LIN {X 0,Y 305.442,Z 224.06,A -85,B 0,C 180,E1 -15871.952,E2 -15871.952} C_VEL
LIN {X 0,Y 305.457,Z 224.06,A -85,B 0,C 180,E1 -15875.114,E2 -15875.114} C_VEL
LIN {X 0,Y 305.461,Z 224.056,A -85,B 0,C 180,E1 -15878.533,E2 -15878.533} C_VEL
LIN {X 0,Y 305.45,Z 224.057,A -85,B 0,C 180,E1 -15882.586,E2 -15882.586} C_VEL
LIN {X 0,Y 305.451,Z 224.223,A -85,B 0,C 180,E1 -15887.041,E2 -15887.041} C_VEL
LIN {X 0,Y 308.59,Z 234.406,A -85,B 0,C 180,E1 -15890.382,E2 -15890.382} C_VEL
LIN {X 0,Y 309.647,Z 238.195,A -85,B 0,C 180,E1 -15891.521,E2 -15891.521} C_VEL
LIN {X 0,Y 318.972,Z 255.957,A -85,B 0,C 180,E1 -15893.321,E2 -15893.321} C_VEL
LIN {X 0,Y 327.178,Z 273.763,A -85,B 0,C 180,E1 -15894.846,E2 -15894.846} C_VEL
LIN {X 0,Y 329.476,Z 279.574,A -85,B 0,C 180,E1 -15895.276,E2 -15895.276} C_VEL
LIN {X 0,Y 331.457,Z 291.54,A -85,B 0,C 180,E1 -15895.818,E2 -15895.818} C_VEL
LIN {X 0,Y 327.97,Z 393.454,A -85,B 0,C 180,E1 -15898.016,E2 -15898.016} C_VEL
LIN {X 0,Y 327.096,Z 410.423,A -85,B 0,C 180,E1 -15898.464,E2 -15898.464} C_VEL
LIN {X 0,Y 325.725,Z 425.453,A -85,B 0,C 180,E1 -15899.084,E2 -15899.084} C_VEL
LIN {X 0,Y 323.988,Z 439.556,A -85,B 0,C 180,E1 -15899.893,E2 -15899.893} C_VEL
LIN {X 0,Y 321.936,Z 453.745,A -85,B 0,C 180,E1 -15900.966,E2 -15900.966} C_VEL
LIN {X 0,Y 319.46,Z 467.76,A -85,B 0,C 180,E1 -15902.307,E2 -15902.307} C_VEL
LIN {X 0,Y 316.903,Z 480.688,A -85,B 0,C 180,E1 -15903.848,E2 -15903.848} C_VEL
LIN {X 0,Y 314.412,Z 492.531,A -85,B 0,C 180,E1 -15905.574,E2 -15905.574} C_VEL
LIN {X 0,Y 311.997,Z 503.387,A -85,B 0,C 180,E1 -15907.485,E2 -15907.485} C_VEL
LIN {X 0,Y 309.684,Z 513.966,A -85,B 0,C 180,E1 -15909.752,E2 -15909.752} C_VEL
LIN {X 0,Y 307.669,Z 522.772,A -85,B 0,C 180,E1 -15912.039,E2 -15912.039} C_VEL
LIN {X 0,Y 306.367,Z 529.155,A -85,B 0,C 180,E1 -15914.022,E2 -15914.022} C_VEL
LIN {X 0,Y 305.081,Z 536.165,A -85,B 0,C 180,E1 -15916.682,E2 -15916.682} C_VEL
LIN {X 0,Y 304.17,Z 541.679,A -85,B 0,C 180,E1 -15919.348,E2 -15919.348} C_VEL
LIN {X 0,Y 303.765,Z 545.855,A -85,B 0,C 180,E1 -15922.021,E2 -15922.021} C_VEL
LIN {X 0,Y 303.596,Z 548.785,A -85,B 0,C 180,E1 -15924.687,E2 -15924.687} C_VEL
LIN {X 0,Y 303.59,Z 550.533,A -85,B 0,C 180,E1 -15927.346,E2 -15927.346} C_VEL
LIN {X 0,Y 303.602,Z 551.13,A -85,B 0,C 180,E1 -15930,E2 -15930} C_VEL
LIN {X 0,Y 303.59,Z 550.523,A -85,B 0,C 180,E1 -15932.654,E2 -15932.654} C_VEL
LIN {X 0,Y 303.624,Z 548.564,A -85,B 0,C 180,E1 -15935.544,E2 -15935.544} C_VEL
LIN {X 0,Y 303.765,Z 545.825,A -85,B 0,C 180,E1 -15937.979,E2 -15937.979} C_VEL
LIN {X 0,Y 304.169,Z 541.644,A -85,B 0,C 180,E1 -15940.652,E2 -15940.652} C_VEL
LIN {X 0,Y 305.068,Z 536.114,A -85,B 0,C 180,E1 -15943.319,E2 -15943.319} C_VEL
LIN {X 0,Y 306.353,Z 529.083,A -85,B 0,C 180,E1 -15945.979,E2 -15945.979} C_VEL
LIN {X 0,Y 308.205,Z 520.343,A -85,B 0,C 180,E1 -15948.617,E2 -15948.617} C_VEL
LIN {X 0,Y 310.329,Z 511.066,A -85,B 0,C 180,E1 -15950.897,E2 -15950.897} C_VEL
LIN {X 0,Y 312.328,Z 501.805,A -85,B 0,C 180,E1 -15952.804,E2 -15952.804} C_VEL
LIN {X 0,Y 314.818,Z 490.441,A -85,B 0,C 180,E1 -15954.744,E2 -15954.744} C_VEL
LIN {X 0,Y 317.361,Z 478.179,A -85,B 0,C 180,E1 -15956.466,E2 -15956.466} C_VEL
LIN {X 0,Y 320.016,Z 464.701,A -85,B 0,C 180,E1 -15957.996,E2 -15957.996} C_VEL
LIN {X 0,Y 322.473,Z 449.936,A -85,B 0,C 180,E1 -15959.336,E2 -15959.336} C_VEL
LIN {X 0,Y 324.543,Z 434.588,A -85,B 0,C 180,E1 -15960.409,E2 -15960.409} C_VEL
LIN {X 0,Y 326.232,Z 419.535,A -85,B 0,C 180,E1 -15961.178,E2 -15961.178} C_VEL
LIN {X 0,Y 327.477,Z 403.763,A -85,B 0,C 180,E1 -15961.721,E2 -15961.721} C_VEL
LIN {X 0,Y 331.104,Z 302.228,A -85,B 0,C 180,E1 -15963.922,E2 -15963.922} C_VEL
LIN {X 0,Y 331.324,Z 291.096,A -85,B 0,C 180,E1 -15964.182,E2 -15964.182} C_VEL
LIN {X 0,Y 328.976,Z 277.875,A -85,B 0,C 180,E1 -15964.8,E2 -15964.8} C_VEL
LIN {X 0,Y 319.974,Z 258.117,A -85,B 0,C 180,E1 -15966.456,E2 -15966.456} C_VEL
LIN {X 0,Y 313.704,Z 245.865,A -85,B 0,C 180,E1 -15967.645,E2 -15967.645} C_VEL
LIN {X 0,Y 309.583,Z 237.999,A -85,B 0,C 180,E1 -15968.468,E2 -15968.468} C_VEL
LIN {X 0,Y 306.264,Z 226.625,A -85,B 0,C 180,E1 -15972.098,E2 -15972.098} C_VEL
LIN {X 0,Y 305.447,Z 224.059,A -85,B 0,C 180,E1 -15972.977,E2 -15972.977} C_VEL
LIN {X 0,Y 305.474,Z 224.053,A -85,B 0,C 180,E1 -15977.409,E2 -15977.409} C_VEL
LIN {X 0,Y 305.504,Z 224.047,A -85,B 0,C 180,E1 -15981.602,E2 -15981.602} C_VEL
LIN {X 0,Y 305.458,Z 224.052,A -85,B 0,C 180,E1 -15984.886,E2 -15984.886} C_VEL
LIN {X 0,Y 305.451,Z 224.059,A -85,B 0,C 180,E1 -15988.353,E2 -15988.353} C_VEL
LIN {X 0,Y 305.523,Z 224.048,A -85,B 0,C 180,E1 -15991.114,E2 -15991.114} C_VEL
LIN {X 0,Y 305.565,Z 224.045,A -85,B 0,C 180,E1 -15994.088,E2 -15994.088} C_VEL
LIN {X 0,Y 305.466,Z 224.029,A -85,B 0,C 180,E1 -15998.4,E2 -15998.4} C_VEL
LIN {X 0,Y 305.583,Z 224.043,A -85,B 0,C 180,E1 -16001.217,E2 -16001.217} C_VEL
LIN {X 0,Y 305.642,Z 224.038,A -85,B 0,C 180,E1 -16005.349,E2 -16005.349} C_VEL
LIN {X 0,Y 305.629,Z 224.041,A -85,B 0,C 180,E1 -16009.4,E2 -16009.4} C_VEL
LIN {X 0,Y 305.79,Z 224.013,A -85,B 0,C 180,E1 -16012.074,E2 -16012.074} C_VEL
LIN {X 0,Y 305.68,Z 224.031,A -85,B 0,C 180,E1 -16014.723,E2 -16014.723} C_VEL
LIN {X 0,Y 305.952,Z 223.998,A -85,B 0,C 180,E1 -16018.684,E2 -16018.684} C_VEL
LIN {X 0,Y 305.952,Z 223.996,A -85,B 0,C 180,E1 -16021.316,E2 -16021.316} C_VEL
LIN {X 0,Y 305.836,Z 224.013,A -85,B 0,C 180,E1 -16026.6,E2 -16026.6} C_VEL
LIN {X 0,Y 305.698,Z 224.024,A -85,B 0,C 180,E1 -16029.261,E2 -16029.261} C_VEL
LIN {X 0,Y 305.582,Z 224.039,A -85,B 0,C 180,E1 -16033.296,E2 -16033.296} C_VEL
LIN {X 0,Y 305.587,Z 224.04,A -85,B 0,C 180,E1 -16036.021,E2 -16036.021} C_VEL
LIN {X 0,Y 305.554,Z 224.047,A -85,B 0,C 180,E1 -16039.436,E2 -16039.436} C_VEL
LIN {X 0,Y 305.481,Z 224.058,A -85,B 0,C 180,E1 -16043.04,E2 -16043.04} C_VEL
LIN {X 0,Y 305.521,Z 224.021,A -85,B 0,C 180,E1 -16046.219,E2 -16046.219} C_VEL
LIN {X 0,Y 305.491,Z 224.057,A -85,B 0,C 180,E1 -16049.051,E2 -16049.051} C_VEL
LIN {X 0,Y 305.46,Z 224.055,A -85,B 0,C 180,E1 -16053.518,E2 -16053.518} C_VEL
LIN {X 0,Y 305.471,Z 224.053,A -85,B 0,C 180,E1 -16056.74,E2 -16056.74} C_VEL
LIN {X 0,Y 305.451,Z 224.059,A -85,B 0,C 180,E1 -16060.6,E2 -16060.6} C_VEL
LIN {X 0,Y 305.416,Z 224.061,A -85,B 0,C 180,E1 -16064.493,E2 -16064.493} C_VEL
LIN {X 0,Y 305.44,Z 224.062,A -85,B 0,C 180,E1 -16068.144,E2 -16068.144} C_VEL
LIN {X 0,Y 305.483,Z 224.145,A -85,B 0,C 180,E1 -16070.766,E2 -16070.766} C_VEL
LIN {X 0,Y 305.611,Z 224.87,A -85,B 0,C 180,E1 -16071.007,E2 -16071.007} C_VEL
LIN {X 0,Y 306.861,Z 227.498,A -85,B 0,C 180,E1 -16071.275,E2 -16071.275} C_VEL
LIN {X 0,Y 309.527,Z 231.534,A -85,B 0,C 180,E1 -16071.79,E2 -16071.79} C_VEL
LIN {X 0,Y 317.49,Z 245.518,A -85,B 0,C 180,E1 -16073.31,E2 -16073.31} C_VEL
LIN {X 0,Y 326.019,Z 262.428,A -85,B 0,C 180,E1 -16074.876,E2 -16074.876} C_VEL
LIN {X 0,Y 331.826,Z 275.27,A -85,B 0,C 180,E1 -16075.915,E2 -16075.915} C_VEL
LIN {X 0,Y 329.059,Z 358.793,A -85,B 0,C 180,E1 -16077.728,E2 -16077.728} C_VEL
LIN {X 0,Y 327.79,Z 390.563,A -85,B 0,C 180,E1 -16078.448,E2 -16078.448} C_VEL
LIN {X 0,Y 326.666,Z 405.546,A -85,B 0,C 180,E1 -16079.012,E2 -16079.012} C_VEL
LIN {X 0,Y 325.15,Z 420.181,A -85,B 0,C 180,E1 -16079.804,E2 -16079.804} C_VEL
LIN {X 0,Y 323.55,Z 433.262,A -85,B 0,C 180,E1 -16080.75,E2 -16080.75} C_VEL
LIN {X 0,Y 321.4,Z 446.754,A -85,B 0,C 180,E1 -16081.958,E2 -16081.958} C_VEL
LIN {X 0,Y 318.907,Z 460.516,A -85,B 0,C 180,E1 -16083.496,E2 -16083.496} C_VEL
LIN {X 0,Y 316.328,Z 473.036,A -85,B 0,C 180,E1 -16085.224,E2 -16085.224} C_VEL
LIN {X 0,Y 314.517,Z 481.644,A -85,B 0,C 180,E1 -16086.652,E2 -16086.652} C_VEL
LIN {X 0,Y 312.254,Z 491.48,A -85,B 0,C 180,E1 -16088.547,E2 -16088.547} C_VEL
LIN {X 0,Y 310.028,Z 501.175,A -85,B 0,C 180,E1 -16090.811,E2 -16090.811} C_VEL
LIN {X 0,Y 308.029,Z 509.515,A -85,B 0,C 180,E1 -16093.177,E2 -16093.177} C_VEL
LIN {X 0,Y 306.709,Z 515.914,A -85,B 0,C 180,E1 -16095.401,E2 -16095.401} C_VEL
LIN {X 0,Y 305.37,Z 522.081,A -85,B 0,C 180,E1 -16098.046,E2 -16098.046} C_VEL
LIN {X 0,Y 304.567,Z 526.836,A -85,B 0,C 180,E1 -16100.705,E2 -16100.705} C_VEL
LIN {X 0,Y 304.046,Z 530.318,A -85,B 0,C 180,E1 -16103.363,E2 -16103.363} C_VEL
LIN {X 0,Y 303.786,Z 532.618,A -85,B 0,C 180,E1 -16106.02,E2 -16106.02} C_VEL
LIN {X 0,Y 303.608,Z 533.793,A -85,B 0,C 180,E1 -16108.674,E2 -16108.674} C_VEL
LIN {X 0,Y 303.608,Z 533.807,A -85,B 0,C 180,E1 -16111.326,E2 -16111.326} C_VEL
LIN {X 0,Y 303.781,Z 532.688,A -85,B 0,C 180,E1 -16113.98,E2 -16113.98} C_VEL
LIN {X 0,Y 304.041,Z 530.442,A -85,B 0,C 180,E1 -16116.637,E2 -16116.637} C_VEL
LIN {X 0,Y 304.551,Z 527.011,A -85,B 0,C 180,E1 -16119.296,E2 -16119.296} C_VEL
LIN {X 0,Y 305.342,Z 522.312,A -85,B 0,C 180,E1 -16121.955,E2 -16121.955} C_VEL
LIN {X 0,Y 306.689,Z 516.215,A -85,B 0,C 180,E1 -16124.6,E2 -16124.6} C_VEL
LIN {X 0,Y 308.303,Z 508.54,A -85,B 0,C 180,E1 -16127.238,E2 -16127.238} C_VEL
LIN {X 0,Y 310.234,Z 500.35,A -85,B 0,C 180,E1 -16129.52,E2 -16129.52} C_VEL
LIN {X 0,Y 312.498,Z 490.48,A -85,B 0,C 180,E1 -16131.782,E2 -16131.782} C_VEL
LIN {X 0,Y 314.726,Z 480.279,A -85,B 0,C 180,E1 -16133.715,E2 -16133.715} C_VEL
LIN {X 0,Y 317.374,Z 468.298,A -85,B 0,C 180,E1 -16135.582,E2 -16135.582} C_VEL
LIN {X 0,Y 319.711,Z 456.205,A -85,B 0,C 180,E1 -16137.137,E2 -16137.137} C_VEL
LIN {X 0,Y 322.091,Z 443.055,A -85,B 0,C 180,E1 -16138.509,E2 -16138.509} C_VEL
LIN {X 0,Y 323.994,Z 429.914,A -85,B 0,C 180,E1 -16139.624,E2 -16139.624} C_VEL
LIN {X 0,Y 325.759,Z 415.327,A -85,B 0,C 180,E1 -16140.589,E2 -16140.589} C_VEL
LIN {X 0,Y 327.093,Z 400.58,A -85,B 0,C 180,E1 -16141.311,E2 -16141.311} C_VEL
LIN {X 0,Y 328.13,Z 385.845,A -85,B 0,C 180,E1 -16141.786,E2 -16141.786} C_VEL
LIN {X 0,Y 331.438,Z 291.969,A -85,B 0,C 180,E1 -16143.82,E2 -16143.82} C_VEL
LIN {X 0,Y 331.228,Z 288.126,A -85,B 0,C 180,E1 -16143.943,E2 -16143.943} C_VEL
LIN {X 0,Y 329.748,Z 282.696,A -85,B 0,C 180,E1 -16144.258,E2 -16144.258} C_VEL
LIN {X 0,Y 327.401,Z 277.728,A -85,B 0,C 180,E1 -16144.67,E2 -16144.67} C_VEL
LIN {X 0,Y 323.608,Z 271.295,A -85,B 0,C 180,E1 -16145.31,E2 -16145.31} C_VEL
LIN {X 0,Y 320.146,Z 264.635,A -85,B 0,C 180,E1 -16145.934,E2 -16145.934} C_VEL
LIN {X 0,Y 311.45,Z 247.476,A -85,B 0,C 180,E1 -16147.599,E2 -16147.599} C_VEL
LIN {X 0,Y 304.686,Z 235.632,A -85,B 0,C 180,E1 -16148.943,E2 -16148.943} C_VEL
LIN {X 0,Y 300.541,Z 229.139,A -85,B 0,C 180,E1 -16149.786,E2 -16149.786} C_VEL
LIN {X 0,Y 298.891,Z 226.755,A -85,B 0,C 180,E1 -16150.126,E2 -16150.126} C_VEL
LIN {X 0,Y 298.433,Z 224.941,A -85,B 0,C 180,E1 -16150.304,E2 -16150.304} C_VEL
LIN {X 0,Y 298.396,Z 224.942,A -85,B 0,C 180,E1 -16153.102,E2 -16153.102} C_VEL
LIN {X 0,Y 298.4,Z 224.925,A -85,B 0,C 180,E1 -16156.92,E2 -16156.92} C_VEL
LIN {X 0,Y 298.421,Z 224.928,A -85,B 0,C 180,E1 -16161,E2 -16161} C_VEL
LIN {X 0,Y 298.428,Z 224.923,A -85,B 0,C 180,E1 -16163.931,E2 -16163.931} C_VEL
LIN {X 0,Y 298.39,Z 224.913,A -85,B 0,C 180,E1 -16167.983,E2 -16167.983} C_VEL
LIN {X 0,Y 298.459,Z 224.933,A -85,B 0,C 180,E1 -16171.904,E2 -16171.904} C_VEL
LIN {X 0,Y 298.48,Z 224.928,A -85,B 0,C 180,E1 -16174.923,E2 -16174.923} C_VEL
LIN {X 0,Y 298.444,Z 224.936,A -85,B 0,C 180,E1 -16179.315,E2 -16179.315} C_VEL
LIN {X 0,Y 298.531,Z 224.916,A -85,B 0,C 180,E1 -16182.179,E2 -16182.179} C_VEL
LIN {X 0,Y 298.587,Z 224.908,A -85,B 0,C 180,E1 -16184.994,E2 -16184.994} C_VEL
LIN {X 0,Y 298.587,Z 224.911,A -85,B 0,C 180,E1 -16189.146,E2 -16189.146} C_VEL
LIN {X 0,Y 298.748,Z 224.895,A -85,B 0,C 180,E1 -16191.886,E2 -16191.886} C_VEL
LIN {X 0,Y 298.651,Z 224.899,A -85,B 0,C 180,E1 -16194.599,E2 -16194.599} C_VEL
LIN {X 0,Y 298.918,Z 224.867,A -85,B 0,C 180,E1 -16198.653,E2 -16198.653} C_VEL
LIN {X 0,Y 298.918,Z 224.875,A -85,B 0,C 180,E1 -16201.347,E2 -16201.347} C_VEL
LIN {X 0,Y 298.78,Z 224.893,A -85,B 0,C 180,E1 -16206.754,E2 -16206.754} C_VEL
LIN {X 0,Y 298.629,Z 224.908,A -85,B 0,C 180,E1 -16209.482,E2 -16209.482} C_VEL
LIN {X 0,Y 298.545,Z 224.916,A -85,B 0,C 180,E1 -16213.616,E2 -16213.616} C_VEL
LIN {X 0,Y 298.542,Z 224.919,A -85,B 0,C 180,E1 -16216.409,E2 -16216.409} C_VEL
LIN {X 0,Y 298.506,Z 224.93,A -85,B 0,C 180,E1 -16219.655,E2 -16219.655} C_VEL
LIN {X 0,Y 298.451,Z 224.936,A -85,B 0,C 180,E1 -16223.598,E2 -16223.598} C_VEL
LIN {X 0,Y 298.484,Z 224.927,A -85,B 0,C 180,E1 -16226.575,E2 -16226.575} C_VEL
LIN {X 0,Y 298.417,Z 224.94,A -85,B 0,C 180,E1 -16229.641,E2 -16229.641} C_VEL
LIN {X 0,Y 298.392,Z 224.932,A -85,B 0,C 180,E1 -16232.8,E2 -16232.8} C_VEL
LIN {X 0,Y 298.446,Z 224.929,A -85,B 0,C 180,E1 -16236.809,E2 -16236.809} C_VEL
LIN {X 0,Y 298.404,Z 224.918,A -85,B 0,C 180,E1 -16239.487,E2 -16239.487} C_VEL
LIN {X 0,Y 298.395,Z 224.942,A -85,B 0,C 180,E1 -16243.104,E2 -16243.104} C_VEL
LIN {X 0,Y 298.394,Z 225.075,A -85,B 0,C 180,E1 -16246.1,E2 -16246.1} C_VEL
LIN {X 0,Y 301.445,Z 234.9,A -85,B 0,C 180,E1 -16249.46,E2 -16249.46} C_VEL
LIN {X 0,Y 302.411,Z 238.056,A -85,B 0,C 180,E1 -16250.426,E2 -16250.426} C_VEL
LIN {X 0,Y 310.708,Z 253.532,A -85,B 0,C 180,E1 -16252.116,E2 -16252.116} C_VEL
LIN {X 0,Y 318.046,Z 268.606,A -85,B 0,C 180,E1 -16253.545,E2 -16253.545} C_VEL
LIN {X 0,Y 323.814,Z 281.919,A -85,B 0,C 180,E1 -16254.645,E2 -16254.645} C_VEL
LIN {X 0,Y 325.566,Z 292.715,A -85,B 0,C 180,E1 -16255.147,E2 -16255.147} C_VEL
LIN {X 0,Y 321.912,Z 395.064,A -85,B 0,C 180,E1 -16257.387,E2 -16257.387} C_VEL
LIN {X 0,Y 320.987,Z 411.376,A -85,B 0,C 180,E1 -16257.838,E2 -16257.838} C_VEL
LIN {X 0,Y 319.482,Z 426.787,A -85,B 0,C 180,E1 -16258.504,E2 -16258.504} C_VEL
LIN {X 0,Y 317.701,Z 440.493,A -85,B 0,C 180,E1 -16259.325,E2 -16259.325} C_VEL
LIN {X 0,Y 315.553,Z 454.674,A -85,B 0,C 180,E1 -16260.438,E2 -16260.438} C_VEL
LIN {X 0,Y 313.181,Z 467.563,A -85,B 0,C 180,E1 -16261.703,E2 -16261.703} C_VEL
LIN {X 0,Y 310.492,Z 480.489,A -85,B 0,C 180,E1 -16263.265,E2 -16263.265} C_VEL
LIN {X 0,Y 307.899,Z 492.331,A -85,B 0,C 180,E1 -16265.022,E2 -16265.022} C_VEL
LIN {X 0,Y 305.281,Z 503.599,A -85,B 0,C 180,E1 -16267.051,E2 -16267.051} C_VEL
LIN {X 0,Y 302.994,Z 513.766,A -85,B 0,C 180,E1 -16269.285,E2 -16269.285} C_VEL
LIN {X 0,Y 300.866,Z 522.572,A -85,B 0,C 180,E1 -16271.619,E2 -16271.619} C_VEL
LIN {X 0,Y 299.142,Z 530.594,A -85,B 0,C 180,E1 -16274.234,E2 -16274.234} C_VEL
LIN {X 0,Y 297.851,Z 537.459,A -85,B 0,C 180,E1 -16277.047,E2 -16277.047} C_VEL
LIN {X 0,Y 296.989,Z 542.647,A -85,B 0,C 180,E1 -16279.777,E2 -16279.777} C_VEL
LIN {X 0,Y 296.691,Z 545.654,A -85,B 0,C 180,E1 -16281.829,E2 -16281.829} C_VEL
LIN {X 0,Y 296.511,Z 548.584,A -85,B 0,C 180,E1 -16284.56,E2 -16284.56} C_VEL
LIN {X 0,Y 296.514,Z 550.332,A -85,B 0,C 180,E1 -16287.283,E2 -16287.283} C_VEL
LIN {X 0,Y 296.517,Z 550.93,A -85,B 0,C 180,E1 -16290,E2 -16290} C_VEL
LIN {X 0,Y 296.514,Z 550.322,A -85,B 0,C 180,E1 -16292.717,E2 -16292.717} C_VEL
LIN {X 0,Y 296.511,Z 548.56,A -85,B 0,C 180,E1 -16295.44,E2 -16295.44} C_VEL
LIN {X 0,Y 296.691,Z 545.622,A -85,B 0,C 180,E1 -16298.171,E2 -16298.171} C_VEL
LIN {X 0,Y 297.131,Z 541.44,A -85,B 0,C 180,E1 -16300.907,E2 -16300.907} C_VEL
LIN {X 0,Y 298.079,Z 535.909,A -85,B 0,C 180,E1 -16303.637,E2 -16303.637} C_VEL
LIN {X 0,Y 299.476,Z 528.879,A -85,B 0,C 180,E1 -16306.356,E2 -16306.356} C_VEL
LIN {X 0,Y 301.409,Z 520.138,A -85,B 0,C 180,E1 -16309.052,E2 -16309.052} C_VEL
LIN {X 0,Y 303.648,Z 510.861,A -85,B 0,C 180,E1 -16311.379,E2 -16311.379} C_VEL
LIN {X 0,Y 305.786,Z 501.431,A -85,B 0,C 180,E1 -16313.357,E2 -16313.357} C_VEL
LIN {X 0,Y 308.572,Z 489.208,A -85,B 0,C 180,E1 -16315.46,E2 -16315.46} C_VEL
LIN {X 0,Y 311.268,Z 476.747,A -85,B 0,C 180,E1 -16317.207,E2 -16317.207} C_VEL
LIN {X 0,Y 313.744,Z 464.495,A -85,B 0,C 180,E1 -16318.607,E2 -16318.607} C_VEL
LIN {X 0,Y 316.096,Z 450.844,A -85,B 0,C 180,E1 -16319.875,E2 -16319.875} C_VEL
LIN {X 0,Y 318.272,Z 435.634,A -85,B 0,C 180,E1 -16320.982,E2 -16320.982} C_VEL
LIN {X 0,Y 320.097,Z 420.216,A -85,B 0,C 180,E1 -16321.798,E2 -16321.798} C_VEL
LIN {X 0,Y 321.386,Z 404.975,A -85,B 0,C 180,E1 -16322.348,E2 -16322.348} C_VEL
LIN {X 0,Y 325.197,Z 303.142,A -85,B 0,C 180,E1 -16324.596,E2 -16324.596} C_VEL
LIN {X 0,Y 325.438,Z 292.247,A -85,B 0,C 180,E1 -16324.852,E2 -16324.852} C_VEL
LIN {X 0,Y 323.35,Z 280.676,A -85,B 0,C 180,E1 -16325.416,E2 -16325.416} C_VEL
LIN {X 0,Y 314.797,Z 261.749,A -85,B 0,C 180,E1 -16327.048,E2 -16327.048} C_VEL
LIN {X 0,Y 308.991,Z 250.246,A -85,B 0,C 180,E1 -16328.19,E2 -16328.19} C_VEL
LIN {X 0,Y 302.262,Z 237.669,A -85,B 0,C 180,E1 -16329.597,E2 -16329.597} C_VEL
LIN {X 0,Y 299.227,Z 227.707,A -85,B 0,C 180,E1 -16332.931,E2 -16332.931} C_VEL
LIN {X 0,Y 298.367,Z 224.945,A -85,B 0,C 180,E1 -16333.955,E2 -16333.955} C_VEL
LIN {X 0,Y 298.399,Z 224.934,A -85,B 0,C 180,E1 -16336.92,E2 -16336.92} C_VEL
LIN {X 0,Y 298.421,Z 224.932,A -85,B 0,C 180,E1 -16341.001,E2 -16341.001} C_VEL
LIN {X 0,Y 298.427,Z 224.927,A -85,B 0,C 180,E1 -16343.932,E2 -16343.932} C_VEL
LIN {X 0,Y 298.394,Z 224.934,A -85,B 0,C 180,E1 -16347.982,E2 -16347.982} C_VEL
LIN {X 0,Y 298.463,Z 224.931,A -85,B 0,C 180,E1 -16351.904,E2 -16351.904} C_VEL
LIN {X 0,Y 298.478,Z 224.93,A -85,B 0,C 180,E1 -16354.924,E2 -16354.924} C_VEL
LIN {X 0,Y 298.431,Z 224.911,A -85,B 0,C 180,E1 -16359.314,E2 -16359.314} C_VEL
LIN {X 0,Y 298.531,Z 224.923,A -85,B 0,C 180,E1 -16362.179,E2 -16362.179} C_VEL
LIN {X 0,Y 298.587,Z 224.914,A -85,B 0,C 180,E1 -16364.995,E2 -16364.995} C_VEL
LIN {X 0,Y 298.585,Z 224.916,A -85,B 0,C 180,E1 -16369.146,E2 -16369.146} C_VEL
LIN {X 0,Y 298.734,Z 224.891,A -85,B 0,C 180,E1 -16371.885,E2 -16371.885} C_VEL
LIN {X 0,Y 298.651,Z 224.907,A -85,B 0,C 180,E1 -16374.599,E2 -16374.599} C_VEL
LIN {X 0,Y 298.918,Z 224.875,A -85,B 0,C 180,E1 -16378.653,E2 -16378.653} C_VEL
LIN {X 0,Y 298.918,Z 224.872,A -85,B 0,C 180,E1 -16381.347,E2 -16381.347} C_VEL
LIN {X 0,Y 298.781,Z 224.893,A -85,B 0,C 180,E1 -16386.754,E2 -16386.754} C_VEL
LIN {X 0,Y 298.629,Z 224.906,A -85,B 0,C 180,E1 -16389.482,E2 -16389.482} C_VEL
LIN {X 0,Y 298.545,Z 224.917,A -85,B 0,C 180,E1 -16393.616,E2 -16393.616} C_VEL
LIN {X 0,Y 298.542,Z 224.916,A -85,B 0,C 180,E1 -16396.409,E2 -16396.409} C_VEL
LIN {X 0,Y 298.492,Z 224.925,A -85,B 0,C 180,E1 -16399.647,E2 -16399.647} C_VEL
LIN {X 0,Y 298.423,Z 224.932,A -85,B 0,C 180,E1 -16403.601,E2 -16403.601} C_VEL
LIN {X 0,Y 298.481,Z 224.899,A -85,B 0,C 180,E1 -16406.575,E2 -16406.575} C_VEL
LIN {X 0,Y 298.416,Z 224.937,A -85,B 0,C 180,E1 -16409.642,E2 -16409.642} C_VEL
LIN {X 0,Y 298.391,Z 224.941,A -85,B 0,C 180,E1 -16412.801,E2 -16412.801} C_VEL
LIN {X 0,Y 298.442,Z 224.928,A -85,B 0,C 180,E1 -16416.808,E2 -16416.808} C_VEL
LIN {X 0,Y 298.384,Z 224.938,A -85,B 0,C 180,E1 -16421.089,E2 -16421.089} C_VEL
LIN {X 0,Y 298.386,Z 224.94,A -85,B 0,C 180,E1 -16425.042,E2 -16425.042} C_VEL
LIN {X 0,Y 298.385,Z 224.943,A -85,B 0,C 180,E1 -16428.913,E2 -16428.913} C_VEL
LIN {X 0,Y 298.435,Z 225.115,A -85,B 0,C 180,E1 -16429.881,E2 -16429.881} C_VEL
LIN {X 0,Y 299.537,Z 227.962,A -85,B 0,C 180,E1 -16430.147,E2 -16430.147} C_VEL
LIN {X 0,Y 301.218,Z 230.109,A -85,B 0,C 180,E1 -16430.481,E2 -16430.481} C_VEL
LIN {X 0,Y 308.701,Z 242.483,A -85,B 0,C 180,E1 -16431.986,E2 -16431.986} C_VEL
LIN {X 0,Y 317.512,Z 259.222,A -85,B 0,C 180,E1 -16433.692,E2 -16433.692} C_VEL
LIN {X 0,Y 325.916,Z 277.372,A -85,B 0,C 180,E1 -16435.258,E2 -16435.258} C_VEL
LIN {X 0,Y 323.813,Z 336.928,A -85,B 0,C 180,E1 -16436.566,E2 -16436.566} C_VEL
LIN {X 0,Y 321.857,Z 389.625,A -85,B 0,C 180,E1 -16437.751,E2 -16437.751} C_VEL
LIN {X 0,Y 320.696,Z 404.902,A -85,B 0,C 180,E1 -16438.319,E2 -16438.319} C_VEL
LIN {X 0,Y 319.093,Z 420.18,A -85,B 0,C 180,E1 -16439.153,E2 -16439.153} C_VEL
LIN {X 0,Y 317.329,Z 433.812,A -85,B 0,C 180,E1 -16440.15,E2 -16440.15} C_VEL
LIN {X 0,Y 314.882,Z 448.515,A -85,B 0,C 180,E1 -16441.506,E2 -16441.506} C_VEL
LIN {X 0,Y 312.3,Z 461.969,A -85,B 0,C 180,E1 -16443.071,E2 -16443.071} C_VEL
LIN {X 0,Y 309.636,Z 474.371,A -85,B 0,C 180,E1 -16444.849,E2 -16444.849} C_VEL
LIN {X 0,Y 307.805,Z 482.665,A -85,B 0,C 180,E1 -16446.276,E2 -16446.276} C_VEL
LIN {X 0,Y 305.245,Z 493.161,A -85,B 0,C 180,E1 -16448.384,E2 -16448.384} C_VEL
LIN {X 0,Y 303.007,Z 502.6,A -85,B 0,C 180,E1 -16450.7,E2 -16450.7} C_VEL
LIN {X 0,Y 300.771,Z 511.387,A -85,B 0,C 180,E1 -16453.342,E2 -16453.342} C_VEL
LIN {X 0,Y 299.452,Z 517.786,A -85,B 0,C 180,E1 -16455.734,E2 -16455.734} C_VEL
LIN {X 0,Y 298.134,Z 523.6,A -85,B 0,C 180,E1 -16458.442,E2 -16458.442} C_VEL
LIN {X 0,Y 297.53,Z 527.038,A -85,B 0,C 180,E1 -16460.483,E2 -16460.483} C_VEL
LIN {X 0,Y 296.999,Z 530.519,A -85,B 0,C 180,E1 -16463.205,E2 -16463.205} C_VEL
LIN {X 0,Y 296.703,Z 532.819,A -85,B 0,C 180,E1 -16465.925,E2 -16465.925} C_VEL
LIN {X 0,Y 296.527,Z 533.994,A -85,B 0,C 180,E1 -16468.642,E2 -16468.642} C_VEL
LIN {X 0,Y 296.527,Z 534.008,A -85,B 0,C 180,E1 -16471.358,E2 -16471.358} C_VEL
LIN {X 0,Y 296.697,Z 532.889,A -85,B 0,C 180,E1 -16474.075,E2 -16474.075} C_VEL
LIN {X 0,Y 296.963,Z 530.643,A -85,B 0,C 180,E1 -16476.796,E2 -16476.796} C_VEL
LIN {X 0,Y 297.516,Z 527.211,A -85,B 0,C 180,E1 -16479.518,E2 -16479.518} C_VEL
LIN {X 0,Y 298.354,Z 522.513,A -85,B 0,C 180,E1 -16482.239,E2 -16482.239} C_VEL
LIN {X 0,Y 299.787,Z 516.415,A -85,B 0,C 180,E1 -16484.944,E2 -16484.944} C_VEL
LIN {X 0,Y 301.479,Z 508.74,A -85,B 0,C 180,E1 -16487.641,E2 -16487.641} C_VEL
LIN {X 0,Y 303.513,Z 500.549,A -85,B 0,C 180,E1 -16489.97,E2 -16489.97} C_VEL
LIN {X 0,Y 305.9,Z 490.679,A -85,B 0,C 180,E1 -16492.276,E2 -16492.276} C_VEL
LIN {X 0,Y 308.205,Z 480.558,A -85,B 0,C 180,E1 -16494.233,E2 -16494.233} C_VEL
LIN {X 0,Y 310.988,Z 468.496,A -85,B 0,C 180,E1 -16496.147,E2 -16496.147} C_VEL
LIN {X 0,Y 313.411,Z 456.401,A -85,B 0,C 180,E1 -16497.729,E2 -16497.729} C_VEL
LIN {X 0,Y 315.874,Z 443.25,A -85,B 0,C 180,E1 -16499.124,E2 -16499.124} C_VEL
LIN {X 0,Y 318.063,Z 428.599,A -85,B 0,C 180,E1 -16500.373,E2 -16500.373} C_VEL
LIN {X 0,Y 319.819,Z 414.091,A -85,B 0,C 180,E1 -16501.321,E2 -16501.321} C_VEL
LIN {X 0,Y 321.248,Z 398.94,A -85,B 0,C 180,E1 -16502.04,E2 -16502.04} C_VEL
LIN {X 0,Y 322.194,Z 384.523,A -85,B 0,C 180,E1 -16502.489,E2 -16502.489} C_VEL
LIN {X 0,Y 326.027,Z 278.846,A -85,B 0,C 180,E1 -16504.809,E2 -16504.809} C_VEL
LIN {X 0,Y 325.833,Z 277.147,A -85,B 0,C 180,E1 -16504.878,E2 -16504.878} C_VEL
LIN {X 0,Y 320.146,Z 264.635,A -85,B 0,C 180,E1 -16505.934,E2 -16505.934} C_VEL
LIN {X 0,Y 318.19,Z 261.752,A -85,B 0,C 180,E1 -16506.271,E2 -16506.271} C_VEL
LIN {X 0,Y 313.718,Z 258.486,A -85,B 0,C 180,E1 -16506.968,E2 -16506.968} C_VEL
LIN {X 0,Y 309.178,Z 255.318,A -85,B 0,C 180,E1 -16507.699,E2 -16507.699} C_VEL
LIN {X 0,Y 307.109,Z 252.561,A -85,B 0,C 180,E1 -16508.081,E2 -16508.081} C_VEL
LIN {X 0,Y 299.236,Z 238.59,A -85,B 0,C 180,E1 -16509.706,E2 -16509.706} C_VEL
LIN {X 0,Y 294.328,Z 231.16,A -85,B 0,C 180,E1 -16510.744,E2 -16510.744} C_VEL
LIN {X 0,Y 291.941,Z 227.88,A -85,B 0,C 180,E1 -16511.256,E2 -16511.256} C_VEL
LIN {X 0,Y 291.331,Z 225.825,A -85,B 0,C 180,E1 -16511.438,E2 -16511.438} C_VEL
LIN {X 0,Y 291.312,Z 225.824,A -85,B 0,C 180,E1 -16515.602,E2 -16515.602} C_VEL
LIN {X 0,Y 291.335,Z 225.817,A -85,B 0,C 180,E1 -16519.358,E2 -16519.358} C_VEL
LIN {X 0,Y 291.424,Z 225.785,A -85,B 0,C 180,E1 -16522.922,E2 -16522.922} C_VEL
LIN {X 0,Y 291.34,Z 225.814,A -85,B 0,C 180,E1 -16526.301,E2 -16526.301} C_VEL
LIN {X 0,Y 291.382,Z 225.799,A -85,B 0,C 180,E1 -16530.26,E2 -16530.26} C_VEL
LIN {X 0,Y 291.411,Z 225.804,A -85,B 0,C 180,E1 -16534.271,E2 -16534.271} C_VEL
LIN {X 0,Y 291.376,Z 225.807,A -85,B 0,C 180,E1 -16537.299,E2 -16537.299} C_VEL
LIN {X 0,Y 291.453,Z 225.804,A -85,B 0,C 180,E1 -16540.27,E2 -16540.27} C_VEL
LIN {X 0,Y 291.535,Z 225.791,A -85,B 0,C 180,E1 -16544.634,E2 -16544.634} C_VEL
LIN {X 0,Y 291.53,Z 225.792,A -85,B 0,C 180,E1 -16548.88,E2 -16548.88} C_VEL
LIN {X 0,Y 291.7,Z 225.773,A -85,B 0,C 180,E1 -16551.688,E2 -16551.688} C_VEL
LIN {X 0,Y 291.622,Z 225.775,A -85,B 0,C 180,E1 -16554.468,E2 -16554.468} C_VEL
LIN {X 0,Y 291.884,Z 225.743,A -85,B 0,C 180,E1 -16558.62,E2 -16558.62} C_VEL
LIN {X 0,Y 291.884,Z 225.751,A -85,B 0,C 180,E1 -16561.38,E2 -16561.38} C_VEL
LIN {X 0,Y 291.729,Z 225.77,A -85,B 0,C 180,E1 -16566.918,E2 -16566.918} C_VEL
LIN {X 0,Y 291.569,Z 225.788,A -85,B 0,C 180,E1 -16569.714,E2 -16569.714} C_VEL
LIN {X 0,Y 291.515,Z 225.793,A -85,B 0,C 180,E1 -16573.95,E2 -16573.95} C_VEL
LIN {X 0,Y 291.481,Z 225.794,A -85,B 0,C 180,E1 -16576.818,E2 -16576.818} C_VEL
LIN {X 0,Y 291.445,Z 225.811,A -85,B 0,C 180,E1 -16579.875,E2 -16579.875} C_VEL
LIN {X 0,Y 291.394,Z 225.813,A -85,B 0,C 180,E1 -16584.206,E2 -16584.206} C_VEL
LIN {X 0,Y 291.417,Z 225.811,A -85,B 0,C 180,E1 -16587.272,E2 -16587.272} C_VEL
LIN {X 0,Y 291.334,Z 225.821,A -85,B 0,C 180,E1 -16590.437,E2 -16590.437} C_VEL
LIN {X 0,Y 291.341,Z 225.814,A -85,B 0,C 180,E1 -16593.699,E2 -16593.699} C_VEL
LIN {X 0,Y 291.379,Z 225.813,A -85,B 0,C 180,E1 -16597.256,E2 -16597.256} C_VEL
LIN {X 0,Y 291.329,Z 225.792,A -85,B 0,C 180,E1 -16600.643,E2 -16600.643} C_VEL
LIN {X 0,Y 291.314,Z 225.821,A -85,B 0,C 180,E1 -16604.912,E2 -16604.912} C_VEL
LIN {X 0,Y 291.323,Z 225.892,A -85,B 0,C 180,E1 -16605.083,E2 -16605.083} C_VEL
LIN {X 0,Y 294.548,Z 236.1,A -85,B 0,C 180,E1 -16608.728,E2 -16608.728} C_VEL
LIN {X 0,Y 294.982,Z 237.621,A -85,B 0,C 180,E1 -16609.217,E2 -16609.217} C_VEL
LIN {X 0,Y 304.88,Z 255.595,A -85,B 0,C 180,E1 -16611.325,E2 -16611.325} C_VEL
LIN {X 0,Y 312.883,Z 272.202,A -85,B 0,C 180,E1 -16612.949,E2 -16612.949} C_VEL
LIN {X 0,Y 318.279,Z 284.898,A -85,B 0,C 180,E1 -16614.021,E2 -16614.021} C_VEL
LIN {X 0,Y 319.74,Z 294.794,A -85,B 0,C 180,E1 -16614.477,E2 -16614.477} C_VEL
LIN {X 0,Y 315.499,Z 404.256,A -85,B 0,C 180,E1 -16616.924,E2 -16616.924} C_VEL
LIN {X 0,Y 314.264,Z 419.663,A -85,B 0,C 180,E1 -16617.493,E2 -16617.493} C_VEL
LIN {X 0,Y 312.373,Z 434.562,A -85,B 0,C 180,E1 -16618.271,E2 -16618.271} C_VEL
LIN {X 0,Y 310.178,Z 449.599,A -85,B 0,C 180,E1 -16619.357,E2 -16619.357} C_VEL
LIN {X 0,Y 307.8,Z 463.001,A -85,B 0,C 180,E1 -16620.6,E2 -16620.6} C_VEL
LIN {X 0,Y 304.921,Z 476.725,A -85,B 0,C 180,E1 -16622.178,E2 -16622.178} C_VEL
LIN {X 0,Y 302.162,Z 489.157,A -85,B 0,C 180,E1 -16623.96,E2 -16623.96} C_VEL
LIN {X 0,Y 299.206,Z 501.349,A -85,B 0,C 180,E1 -16626.098,E2 -16626.098} C_VEL
LIN {X 0,Y 296.632,Z 512.203,A -85,B 0,C 180,E1 -16628.455,E2 -16628.455} C_VEL
LIN {X 0,Y 294.339,Z 521.244,A -85,B 0,C 180,E1 -16630.834,E2 -16630.834} C_VEL
LIN {X 0,Y 292.6,Z 528.752,A -85,B 0,C 180,E1 -16633.248,E2 -16633.248} C_VEL
LIN {X 0,Y 291.123,Z 535.761,A -85,B 0,C 180,E1 -16636.031,E2 -16636.031} C_VEL
LIN {X 0,Y 290.107,Z 541.276,A -85,B 0,C 180,E1 -16638.825,E2 -16638.825} C_VEL
LIN {X 0,Y 289.613,Z 545.452,A -85,B 0,C 180,E1 -16641.628,E2 -16641.628} C_VEL
LIN {X 0,Y 289.426,Z 548.534,A -85,B 0,C 180,E1 -16644.611,E2 -16644.611} C_VEL
LIN {X 0,Y 289.417,Z 550.132,A -85,B 0,C 180,E1 -16647.216,E2 -16647.216} C_VEL
LIN {X 0,Y 289.434,Z 550.729,A -85,B 0,C 180,E1 -16650,E2 -16650} C_VEL
LIN {X 0,Y 289.417,Z 550.121,A -85,B 0,C 180,E1 -16652.784,E2 -16652.784} C_VEL
LIN {X 0,Y 289.432,Z 548.359,A -85,B 0,C 180,E1 -16655.574,E2 -16655.574} C_VEL
LIN {X 0,Y 289.613,Z 545.419,A -85,B 0,C 180,E1 -16658.372,E2 -16658.372} C_VEL
LIN {X 0,Y 290.106,Z 541.237,A -85,B 0,C 180,E1 -16661.175,E2 -16661.175} C_VEL
LIN {X 0,Y 291.106,Z 535.705,A -85,B 0,C 180,E1 -16663.97,E2 -16663.97} C_VEL
LIN {X 0,Y 292.599,Z 528.674,A -85,B 0,C 180,E1 -16666.752,E2 -16666.752} C_VEL
LIN {X 0,Y 294.634,Z 519.933,A -85,B 0,C 180,E1 -16669.508,E2 -16669.508} C_VEL
LIN {X 0,Y 296.984,Z 510.656,A -85,B 0,C 180,E1 -16671.883,E2 -16671.883} C_VEL
LIN {X 0,Y 299.213,Z 501.226,A -85,B 0,C 180,E1 -16673.901,E2 -16673.901} C_VEL
LIN {X 0,Y 302.13,Z 489.002,A -85,B 0,C 180,E1 -16676.043,E2 -16676.043} C_VEL
LIN {X 0,Y 304.915,Z 476.54,A -85,B 0,C 180,E1 -16677.822,E2 -16677.822} C_VEL
LIN {X 0,Y 307.787,Z 462.757,A -85,B 0,C 180,E1 -16679.401,E2 -16679.401} C_VEL
LIN {X 0,Y 310.158,Z 449.372,A -85,B 0,C 180,E1 -16680.637,E2 -16680.637} C_VEL
LIN {X 0,Y 312.357,Z 434.171,A -85,B 0,C 180,E1 -16681.73,E2 -16681.73} C_VEL
LIN {X 0,Y 314.169,Z 419.112,A -85,B 0,C 180,E1 -16682.518,E2 -16682.518} C_VEL
LIN {X 0,Y 315.489,Z 403.325,A -85,B 0,C 180,E1 -16683.077,E2 -16683.077} C_VEL
LIN {X 0,Y 319.579,Z 296.916,A -85,B 0,C 180,E1 -16685.455,E2 -16685.455} C_VEL
LIN {X 0,Y 319.433,Z 292.676,A -85,B 0,C 180,E1 -16685.588,E2 -16685.588} C_VEL
LIN {X 0,Y 317.887,Z 283.722,A -85,B 0,C 180,E1 -16686.03,E2 -16686.03} C_VEL
LIN {X 0,Y 309.636,Z 265.317,A -85,B 0,C 180,E1 -16687.664,E2 -16687.664} C_VEL
LIN {X 0,Y 303.822,Z 253.735,A -85,B 0,C 180,E1 -16688.851,E2 -16688.851} C_VEL
LIN {X 0,Y 296.976,Z 241.309,A -85,B 0,C 180,E1 -16690.298,E2 -16690.298} C_VEL
LIN {X 0,Y 294.865,Z 237.314,A -85,B 0,C 180,E1 -16690.822,E2 -16690.822} C_VEL
LIN {X 0,Y 292.202,Z 228.776,A -85,B 0,C 180,E1 -16693.817,E2 -16693.817} C_VEL
LIN {X 0,Y 291.322,Z 225.817,A -85,B 0,C 180,E1 -16694.923,E2 -16694.923} C_VEL
LIN {X 0,Y 291.37,Z 225.807,A -85,B 0,C 180,E1 -16699.364,E2 -16699.364} C_VEL
LIN {X 0,Y 291.424,Z 225.803,A -85,B 0,C 180,E1 -16702.922,E2 -16702.922} C_VEL
LIN {X 0,Y 291.341,Z 225.812,A -85,B 0,C 180,E1 -16706.301,E2 -16706.301} C_VEL
LIN {X 0,Y 291.385,Z 225.805,A -85,B 0,C 180,E1 -16710.259,E2 -16710.259} C_VEL
LIN {X 0,Y 291.411,Z 225.809,A -85,B 0,C 180,E1 -16714.272,E2 -16714.272} C_VEL
LIN {X 0,Y 291.365,Z 225.79,A -85,B 0,C 180,E1 -16717.298,E2 -16717.298} C_VEL
LIN {X 0,Y 291.452,Z 225.793,A -85,B 0,C 180,E1 -16720.27,E2 -16720.27} C_VEL
LIN {X 0,Y 291.535,Z 225.792,A -85,B 0,C 180,E1 -16724.634,E2 -16724.634} C_VEL
LIN {X 0,Y 291.529,Z 225.793,A -85,B 0,C 180,E1 -16728.88,E2 -16728.88} C_VEL
LIN {X 0,Y 291.681,Z 225.769,A -85,B 0,C 180,E1 -16731.688,E2 -16731.688} C_VEL
LIN {X 0,Y 291.621,Z 225.783,A -85,B 0,C 180,E1 -16734.468,E2 -16734.468} C_VEL
LIN {X 0,Y 291.884,Z 225.751,A -85,B 0,C 180,E1 -16738.62,E2 -16738.62} C_VEL
LIN {X 0,Y 291.885,Z 225.748,A -85,B 0,C 180,E1 -16741.38,E2 -16741.38} C_VEL
LIN {X 0,Y 291.73,Z 225.772,A -85,B 0,C 180,E1 -16746.918,E2 -16746.918} C_VEL
LIN {X 0,Y 291.569,Z 225.787,A -85,B 0,C 180,E1 -16749.714,E2 -16749.714} C_VEL
LIN {X 0,Y 291.516,Z 225.796,A -85,B 0,C 180,E1 -16753.951,E2 -16753.951} C_VEL
LIN {X 0,Y 291.48,Z 225.794,A -85,B 0,C 180,E1 -16756.818,E2 -16756.818} C_VEL
LIN {X 0,Y 291.446,Z 225.802,A -85,B 0,C 180,E1 -16759.875,E2 -16759.875} C_VEL
LIN {X 0,Y 291.377,Z 225.801,A -85,B 0,C 180,E1 -16764.208,E2 -16764.208} C_VEL
LIN {X 0,Y 291.416,Z 225.785,A -85,B 0,C 180,E1 -16767.272,E2 -16767.272} C_VEL
LIN {X 0,Y 291.333,Z 225.817,A -85,B 0,C 180,E1 -16770.438,E2 -16770.438} C_VEL
LIN {X 0,Y 291.34,Z 225.812,A -85,B 0,C 180,E1 -16773.699,E2 -16773.699} C_VEL
LIN {X 0,Y 291.372,Z 225.809,A -85,B 0,C 180,E1 -16777.255,E2 -16777.255} C_VEL
LIN {X 0,Y 291.33,Z 225.818,A -85,B 0,C 180,E1 -16780.643,E2 -16780.643} C_VEL
LIN {X 0,Y 291.311,Z 225.818,A -85,B 0,C 180,E1 -16784.398,E2 -16784.398} C_VEL
LIN {X 0,Y 291.364,Z 225.857,A -85,B 0,C 180,E1 -16788.714,E2 -16788.714} C_VEL
LIN {X 0,Y 292.339,Z 228.662,A -85,B 0,C 180,E1 -16788.972,E2 -16788.972} C_VEL
LIN {X 0,Y 294.278,Z 231.081,A -85,B 0,C 180,E1 -16789.379,E2 -16789.379} C_VEL
LIN {X 0,Y 296.494,Z 234.41,A -85,B 0,C 180,E1 -16789.852,E2 -16789.852} C_VEL
LIN {X 0,Y 303.981,Z 246.783,A -85,B 0,C 180,E1 -16791.41,E2 -16791.41} C_VEL
LIN {X 0,Y 312.631,Z 263.453,A -85,B 0,C 180,E1 -16793.145,E2 -16793.145} C_VEL
LIN {X 0,Y 320.026,Z 279.442,A -85,B 0,C 180,E1 -16794.573,E2 -16794.573} C_VEL
LIN {X 0,Y 318.036,Z 335.007,A -85,B 0,C 180,E1 -16795.819,E2 -16795.819} C_VEL
LIN {X 0,Y 315.895,Z 389.842,A -85,B 0,C 180,E1 -16797.066,E2 -16797.066} C_VEL
LIN {X 0,Y 314.683,Z 405.114,A -85,B 0,C 180,E1 -16797.641,E2 -16797.641} C_VEL
LIN {X 0,Y 313.033,Z 420.388,A -85,B 0,C 180,E1 -16798.488,E2 -16798.488} C_VEL
LIN {X 0,Y 311.145,Z 434.347,A -85,B 0,C 180,E1 -16799.526,E2 -16799.526} C_VEL
LIN {X 0,Y 308.675,Z 448.721,A -85,B 0,C 180,E1 -16800.879,E2 -16800.879} C_VEL
LIN {X 0,Y 305.985,Z 462.174,A -85,B 0,C 180,E1 -16802.469,E2 -16802.469} C_VEL
LIN {X 0,Y 303.23,Z 474.381,A -85,B 0,C 180,E1 -16804.243,E2 -16804.243} C_VEL
LIN {X 0,Y 301.197,Z 483.277,A -85,B 0,C 180,E1 -16805.807,E2 -16805.807} C_VEL
LIN {X 0,Y 298.622,Z 493.365,A -85,B 0,C 180,E1 -16807.88,E2 -16807.88} C_VEL
LIN {X 0,Y 296.269,Z 502.805,A -85,B 0,C 180,E1 -16810.243,E2 -16810.243} C_VEL
LIN {X 0,Y 294.19,Z 510.665,A -85,B 0,C 180,E1 -16812.627,E2 -16812.627} C_VEL
LIN {X 0,Y 292.537,Z 517.989,A -85,B 0,C 180,E1 -16815.389,E2 -16815.389} C_VEL
LIN {X 0,Y 291.151,Z 523.803,A -85,B 0,C 180,E1 -16818.16,E2 -16818.16} C_VEL
LIN {X 0,Y 290.515,Z 527.24,A -85,B 0,C 180,E1 -16820.251,E2 -16820.251} C_VEL
LIN {X 0,Y 289.948,Z 530.721,A -85,B 0,C 180,E1 -16823.039,E2 -16823.039} C_VEL
LIN {X 0,Y 289.623,Z 533.02,A -85,B 0,C 180,E1 -16825.825,E2 -16825.825} C_VEL
LIN {X 0,Y 289.448,Z 534.194,A -85,B 0,C 180,E1 -16828.609,E2 -16828.609} C_VEL
LIN {X 0,Y 289.448,Z 534.208,A -85,B 0,C 180,E1 -16831.391,E2 -16831.391} C_VEL
LIN {X 0,Y 289.616,Z 533.089,A -85,B 0,C 180,E1 -16834.175,E2 -16834.175} C_VEL
LIN {X 0,Y 289.889,Z 530.844,A -85,B 0,C 180,E1 -16836.962,E2 -16836.962} C_VEL
LIN {X 0,Y 290.503,Z 527.412,A -85,B 0,C 180,E1 -16839.75,E2 -16839.75} C_VEL
LIN {X 0,Y 291.379,Z 522.714,A -85,B 0,C 180,E1 -16842.537,E2 -16842.537} C_VEL
LIN {X 0,Y 292.893,Z 516.616,A -85,B 0,C 180,E1 -16845.304,E2 -16845.304} C_VEL
LIN {X 0,Y 294.677,Z 508.941,A -85,B 0,C 180,E1 -16848.062,E2 -16848.062} C_VEL
LIN {X 0,Y 296.816,Z 500.749,A -85,B 0,C 180,E1 -16850.441,E2 -16850.441} C_VEL
LIN {X 0,Y 299.335,Z 490.877,A -85,B 0,C 180,E1 -16852.792,E2 -16852.792} C_VEL
LIN {X 0,Y 301.742,Z 480.756,A -85,B 0,C 180,E1 -16854.786,E2 -16854.786} C_VEL
LIN {X 0,Y 304.638,Z 468.693,A -85,B 0,C 180,E1 -16856.734,E2 -16856.734} C_VEL
LIN {X 0,Y 307.119,Z 456.598,A -85,B 0,C 180,E1 -16858.348,E2 -16858.348} C_VEL
LIN {X 0,Y 309.678,Z 443.446,A -85,B 0,C 180,E1 -16859.764,E2 -16859.764} C_VEL
LIN {X 0,Y 311.763,Z 430.168,A -85,B 0,C 180,E1 -16860.923,E2 -16860.923} C_VEL
LIN {X 0,Y 313.62,Z 415.71,A -85,B 0,C 180,E1 -16861.909,E2 -16861.909} C_VEL
LIN {X 0,Y 315.084,Z 400.956,A -85,B 0,C 180,E1 -16862.649,E2 -16862.649} C_VEL
LIN {X 0,Y 316.187,Z 386.205,A -85,B 0,C 180,E1 -16863.137,E2 -16863.137} C_VEL
LIN {X 0,Y 320.133,Z 281.108,A -85,B 0,C 180,E1 -16865.489,E2 -16865.489} C_VEL
LIN {X 0,Y 319.957,Z 279.217,A -85,B 0,C 180,E1 -16865.563,E2 -16865.563} C_VEL
LIN {X 0,Y 311.936,Z 261.99,A -85,B 0,C 180,E1 -16867.117,E2 -16867.117} C_VEL
LIN {X 0,Y 307.109,Z 252.561,A -85,B 0,C 180,E1 -16868.081,E2 -16868.081} C_VEL
LIN {X 0,Y 304.275,Z 248.322,A -85,B 0,C 180,E1 -16868.628,E2 -16868.628} C_VEL
LIN {X 0,Y 300.787,Z 244.916,A -85,B 0,C 180,E1 -16869.268,E2 -16869.268} C_VEL
LIN {X 0,Y 290.869,Z 236.904,A -85,B 0,C 180,E1 -16871.152,E2 -16871.152} C_VEL
LIN {X 0,Y 288.721,Z 234.433,A -85,B 0,C 180,E1 -16871.608,E2 -16871.608} C_VEL
LIN {X 0,Y 286.792,Z 231.297,A -85,B 0,C 180,E1 -16872.057,E2 -16872.057} C_VEL
LIN {X 0,Y 284.889,Z 228.822,A -85,B 0,C 180,E1 -16872.489,E2 -16872.489} C_VEL
LIN {X 0,Y 284.277,Z 226.699,A -85,B 0,C 180,E1 -16872.695,E2 -16872.695} C_VEL
LIN {X 0,Y 284.266,Z 226.692,A -85,B 0,C 180,E1 -16876.191,E2 -16876.191} C_VEL
LIN {X 0,Y 284.308,Z 226.696,A -85,B 0,C 180,E1 -16880.022,E2 -16880.022} C_VEL
LIN {X 0,Y 284.348,Z 226.671,A -85,B 0,C 180,E1 -16883.616,E2 -16883.616} C_VEL
LIN {X 0,Y 284.303,Z 226.675,A -85,B 0,C 180,E1 -16887.189,E2 -16887.189} C_VEL
LIN {X 0,Y 284.354,Z 226.676,A -85,B 0,C 180,E1 -16890.375,E2 -16890.375} C_VEL
LIN {X 0,Y 284.373,Z 226.679,A -85,B 0,C 180,E1 -16893.586,E2 -16893.586} C_VEL
LIN {X 0,Y 284.361,Z 226.683,A -85,B 0,C 180,E1 -16896.706,E2 -16896.706} C_VEL
LIN {X 0,Y 284.397,Z 226.675,A -85,B 0,C 180,E1 -16901.261,E2 -16901.261} C_VEL
LIN {X 0,Y 284.473,Z 226.672,A -85,B 0,C 180,E1 -16904.469,E2 -16904.469} C_VEL
LIN {X 0,Y 284.482,Z 226.673,A -85,B 0,C 180,E1 -16908.601,E2 -16908.601} C_VEL
LIN {X 0,Y 284.651,Z 226.65,A -85,B 0,C 180,E1 -16911.481,E2 -16911.481} C_VEL
LIN {X 0,Y 284.592,Z 226.65,A -85,B 0,C 180,E1 -16914.331,E2 -16914.331} C_VEL
LIN {X 0,Y 284.85,Z 226.619,A -85,B 0,C 180,E1 -16918.586,E2 -16918.586} C_VEL
LIN {X 0,Y 284.85,Z 226.628,A -85,B 0,C 180,E1 -16921.414,E2 -16921.414} C_VEL
LIN {X 0,Y 284.68,Z 226.647,A -85,B 0,C 180,E1 -16927.09,E2 -16927.09} C_VEL
LIN {X 0,Y 284.513,Z 226.668,A -85,B 0,C 180,E1 -16929.957,E2 -16929.957} C_VEL
LIN {X 0,Y 284.472,Z 226.673,A -85,B 0,C 180,E1 -16934.303,E2 -16934.303} C_VEL
LIN {X 0,Y 284.419,Z 226.672,A -85,B 0,C 180,E1 -16937.249,E2 -16937.249} C_VEL
LIN {X 0,Y 284.373,Z 226.688,A -85,B 0,C 180,E1 -16940.242,E2 -16940.242} C_VEL
LIN {X 0,Y 284.364,Z 226.693,A -85,B 0,C 180,E1 -16943.876,E2 -16943.876} C_VEL
LIN {X 0,Y 284.392,Z 226.687,A -85,B 0,C 180,E1 -16947.174,E2 -16947.174} C_VEL
LIN {X 0,Y 284.293,Z 226.698,A -85,B 0,C 180,E1 -16951.274,E2 -16951.274} C_VEL
LIN {X 0,Y 284.337,Z 226.689,A -85,B 0,C 180,E1 -16955.349,E2 -16955.349} C_VEL
LIN {X 0,Y 284.315,Z 226.693,A -85,B 0,C 180,E1 -16958.168,E2 -16958.168} C_VEL
LIN {X 0,Y 284.264,Z 226.685,A -85,B 0,C 180,E1 -16962.125,E2 -16962.125} C_VEL
LIN {X 0,Y 284.252,Z 226.743,A -85,B 0,C 180,E1 -16964.01,E2 -16964.01} C_VEL
LIN {X 0,Y 287.704,Z 237.476,A -85,B 0,C 180,E1 -16967.957,E2 -16967.957} C_VEL
LIN {X 0,Y 296.323,Z 252.766,A -85,B 0,C 180,E1 -16969.909,E2 -16969.909} C_VEL
LIN {X 0,Y 304.066,Z 267.82,A -85,B 0,C 180,E1 -16971.564,E2 -16971.564} C_VEL
LIN {X 0,Y 311.76,Z 285.035,A -85,B 0,C 180,E1 -16973.156,E2 -16973.156} C_VEL
LIN {X 0,Y 312.803,Z 287.959,A -85,B 0,C 180,E1 -16973.38,E2 -16973.38} C_VEL
LIN {X 0,Y 313.915,Z 295.926,A -85,B 0,C 180,E1 -16973.751,E2 -16973.751} C_VEL
LIN {X 0,Y 309.652,Z 402.574,A -85,B 0,C 180,E1 -16976.168,E2 -16976.168} C_VEL
LIN {X 0,Y 308.468,Z 417.644,A -85,B 0,C 180,E1 -16976.707,E2 -16976.707} C_VEL
LIN {X 0,Y 306.523,Z 433.066,A -85,B 0,C 180,E1 -16977.496,E2 -16977.496} C_VEL
LIN {X 0,Y 304.411,Z 447.317,A -85,B 0,C 180,E1 -16978.509,E2 -16978.509} C_VEL
LIN {X 0,Y 301.931,Z 461.22,A -85,B 0,C 180,E1 -16979.778,E2 -16979.778} C_VEL
LIN {X 0,Y 299.229,Z 473.939,A -85,B 0,C 180,E1 -16981.218,E2 -16981.218} C_VEL
LIN {X 0,Y 296.249,Z 486.811,A -85,B 0,C 180,E1 -16983.019,E2 -16983.019} C_VEL
LIN {X 0,Y 293.539,Z 497.591,A -85,B 0,C 180,E1 -16984.852,E2 -16984.852} C_VEL
LIN {X 0,Y 291.02,Z 507.562,A -85,B 0,C 180,E1 -16986.892,E2 -16986.892} C_VEL
LIN {X 0,Y 288.881,Z 516.086,A -85,B 0,C 180,E1 -16988.971,E2 -16988.971} C_VEL
LIN {X 0,Y 286.698,Z 524.418,A -85,B 0,C 180,E1 -16991.418,E2 -16991.418} C_VEL
LIN {X 0,Y 284.908,Z 532.254,A -85,B 0,C 180,E1 -16994.256,E2 -16994.256} C_VEL
LIN {X 0,Y 283.616,Z 538.494,A -85,B 0,C 180,E1 -16997.114,E2 -16997.114} C_VEL
LIN {X 0,Y 282.767,Z 543.323,A -85,B 0,C 180,E1 -16999.981,E2 -16999.981} C_VEL
LIN {X 0,Y 282.386,Z 546.867,A -85,B 0,C 180,E1 -17002.852,E2 -17002.852} C_VEL
LIN {X 0,Y 282.285,Z 549.2,A -85,B 0,C 180,E1 -17005.717,E2 -17005.717} C_VEL
LIN {X 0,Y 282.332,Z 550.374,A -85,B 0,C 180,E1 -17008.574,E2 -17008.574} C_VEL
LIN {X 0,Y 282.332,Z 550.371,A -85,B 0,C 180,E1 -17011.426,E2 -17011.426} C_VEL
LIN {X 0,Y 282.285,Z 549.182,A -85,B 0,C 180,E1 -17014.283,E2 -17014.283} C_VEL
LIN {X 0,Y 282.386,Z 546.836,A -85,B 0,C 180,E1 -17017.148,E2 -17017.148} C_VEL
LIN {X 0,Y 282.767,Z 543.286,A -85,B 0,C 180,E1 -17020.019,E2 -17020.019} C_VEL
LIN {X 0,Y 283.61,Z 538.446,A -85,B 0,C 180,E1 -17022.886,E2 -17022.886} C_VEL
LIN {X 0,Y 284.752,Z 532.18,A -85,B 0,C 180,E1 -17025.753,E2 -17025.753} C_VEL
LIN {X 0,Y 286.699,Z 524.329,A -85,B 0,C 180,E1 -17028.582,E2 -17028.582} C_VEL
LIN {X 0,Y 288.883,Z 515.985,A -85,B 0,C 180,E1 -17031.028,E2 -17031.028} C_VEL
LIN {X 0,Y 291.329,Z 506.126,A -85,B 0,C 180,E1 -17033.41,E2 -17033.41} C_VEL
LIN {X 0,Y 294.03,Z 495.665,A -85,B 0,C 180,E1 -17035.482,E2 -17035.482} C_VEL
LIN {X 0,Y 297.017,Z 483.429,A -85,B 0,C 180,E1 -17037.477,E2 -17037.477} C_VEL
LIN {X 0,Y 299.773,Z 471.151,A -85,B 0,C 180,E1 -17039.108,E2 -17039.108} C_VEL
LIN {X 0,Y 302.513,Z 457.79,A -85,B 0,C 180,E1 -17040.543,E2 -17040.543} C_VEL
LIN {X 0,Y 305.078,Z 443.042,A -85,B 0,C 180,E1 -17041.8,E2 -17041.8} C_VEL
LIN {X 0,Y 307.031,Z 428.756,A -85,B 0,C 180,E1 -17042.736,E2 -17042.736} C_VEL
LIN {X 0,Y 308.78,Z 413.399,A -85,B 0,C 180,E1 -17043.451,E2 -17043.451} C_VEL
LIN {X 0,Y 309.81,Z 398.585,A -85,B 0,C 180,E1 -17043.91,E2 -17043.91} C_VEL
LIN {X 0,Y 313.84,Z 295.674,A -85,B 0,C 180,E1 -17046.233,E2 -17046.233} C_VEL
LIN {X 0,Y 312.411,Z 286.666,A -85,B 0,C 180,E1 -17046.675,E2 -17046.675} C_VEL
LIN {X 0,Y 304.171,Z 268.086,A -85,B 0,C 180,E1 -17048.375,E2 -17048.375} C_VEL
LIN {X 0,Y 295.632,Z 251.368,A -85,B 0,C 180,E1 -17050.205,E2 -17050.205} C_VEL
LIN {X 0,Y 289.368,Z 240.567,A -85,B 0,C 180,E1 -17051.602,E2 -17051.602} C_VEL
LIN {X 0,Y 287.591,Z 237.19,A -85,B 0,C 180,E1 -17052.041,E2 -17052.041} C_VEL
LIN {X 0,Y 284.27,Z 226.7,A -85,B 0,C 180,E1 -17055.99,E2 -17055.99} C_VEL
LIN {X 0,Y 284.347,Z 226.684,A -85,B 0,C 180,E1 -17060.013,E2 -17060.013} C_VEL
LIN {X 0,Y 284.348,Z 226.683,A -85,B 0,C 180,E1 -17063.617,E2 -17063.617} C_VEL
LIN {X 0,Y 284.304,Z 226.685,A -85,B 0,C 180,E1 -17067.189,E2 -17067.189} C_VEL
LIN {X 0,Y 284.357,Z 226.681,A -85,B 0,C 180,E1 -17070.376,E2 -17070.376} C_VEL
LIN {X 0,Y 284.373,Z 226.68,A -85,B 0,C 180,E1 -17073.586,E2 -17073.586} C_VEL
LIN {X 0,Y 284.327,Z 226.674,A -85,B 0,C 180,E1 -17076.704,E2 -17076.704} C_VEL
LIN {X 0,Y 284.397,Z 226.682,A -85,B 0,C 180,E1 -17081.261,E2 -17081.261} C_VEL
LIN {X 0,Y 284.472,Z 226.671,A -85,B 0,C 180,E1 -17084.47,E2 -17084.47} C_VEL
LIN {X 0,Y 284.481,Z 226.671,A -85,B 0,C 180,E1 -17088.601,E2 -17088.601} C_VEL
LIN {X 0,Y 284.632,Z 226.647,A -85,B 0,C 180,E1 -17091.48,E2 -17091.48} C_VEL
LIN {X 0,Y 284.591,Z 226.658,A -85,B 0,C 180,E1 -17094.331,E2 -17094.331} C_VEL
LIN {X 0,Y 284.85,Z 226.627,A -85,B 0,C 180,E1 -17098.586,E2 -17098.586} C_VEL
LIN {X 0,Y 284.85,Z 226.625,A -85,B 0,C 180,E1 -17101.414,E2 -17101.414} C_VEL
LIN {X 0,Y 284.681,Z 226.649,A -85,B 0,C 180,E1 -17107.091,E2 -17107.091} C_VEL
LIN {X 0,Y 284.513,Z 226.669,A -85,B 0,C 180,E1 -17109.957,E2 -17109.957} C_VEL
LIN {X 0,Y 284.472,Z 226.673,A -85,B 0,C 180,E1 -17114.303,E2 -17114.303} C_VEL
LIN {X 0,Y 284.417,Z 226.675,A -85,B 0,C 180,E1 -17117.249,E2 -17117.249} C_VEL
LIN {X 0,Y 284.372,Z 226.681,A -85,B 0,C 180,E1 -17120.243,E2 -17120.243} C_VEL
LIN {X 0,Y 284.331,Z 226.667,A -85,B 0,C 180,E1 -17124.847,E2 -17124.847} C_VEL
LIN {X 0,Y 284.326,Z 226.68,A -85,B 0,C 180,E1 -17128.011,E2 -17128.011} C_VEL
LIN {X 0,Y 284.291,Z 226.693,A -85,B 0,C 180,E1 -17131.275,E2 -17131.275} C_VEL
LIN {X 0,Y 284.337,Z 226.691,A -85,B 0,C 180,E1 -17135.349,E2 -17135.349} C_VEL
LIN {X 0,Y 284.308,Z 226.693,A -85,B 0,C 180,E1 -17138.17,E2 -17138.17} C_VEL
LIN {X 0,Y 284.266,Z 226.693,A -85,B 0,C 180,E1 -17142.125,E2 -17142.125} C_VEL
LIN {X 0,Y 284.266,Z 226.697,A -85,B 0,C 180,E1 -17146.193,E2 -17146.193} C_VEL
LIN {X 0,Y 284.291,Z 226.834,A -85,B 0,C 180,E1 -17147.472,E2 -17147.472} C_VEL
LIN {X 0,Y 285.219,Z 229.466,A -85,B 0,C 180,E1 -17147.732,E2 -17147.732} C_VEL
LIN {X 0,Y 287.307,Z 232.012,A -85,B 0,C 180,E1 -17148.197,E2 -17148.197} C_VEL
LIN {X 0,Y 289.487,Z 235.356,A -85,B 0,C 180,E1 -17148.693,E2 -17148.693} C_VEL
LIN {X 0,Y 296.951,Z 247.006,A -85,B 0,C 180,E1 -17150.317,E2 -17150.317} C_VEL
LIN {X 0,Y 304.972,Z 261.937,A -85,B 0,C 180,E1 -17152.006,E2 -17152.006} C_VEL
LIN {X 0,Y 312.943,Z 278.779,A -85,B 0,C 180,E1 -17153.619,E2 -17153.619} C_VEL
LIN {X 0,Y 314.28,Z 281.844,A -85,B 0,C 180,E1 -17153.885,E2 -17153.885} C_VEL
LIN {X 0,Y 309.976,Z 390.059,A -85,B 0,C 180,E1 -17156.355,E2 -17156.355} C_VEL
LIN {X 0,Y 308.718,Z 405.326,A -85,B 0,C 180,E1 -17156.937,E2 -17156.937} C_VEL
LIN {X 0,Y 307.009,Z 420.597,A -85,B 0,C 180,E1 -17157.796,E2 -17157.796} C_VEL
LIN {X 0,Y 305.002,Z 434.863,A -85,B 0,C 180,E1 -17158.876,E2 -17158.876} C_VEL
LIN {X 0,Y 302.501,Z 448.926,A -85,B 0,C 180,E1 -17160.225,E2 -17160.225} C_VEL
LIN {X 0,Y 299.707,Z 462.379,A -85,B 0,C 180,E1 -17161.842,E2 -17161.842} C_VEL
LIN {X 0,Y 296.853,Z 474.585,A -85,B 0,C 180,E1 -17163.647,E2 -17163.647} C_VEL
LIN {X 0,Y 294.789,Z 482.929,A -85,B 0,C 180,E1 -17165.128,E2 -17165.128} C_VEL
LIN {X 0,Y 292.463,Z 492.092,A -85,B 0,C 180,E1 -17167.015,E2 -17167.015} C_VEL
LIN {X 0,Y 289.869,Z 501.788,A -85,B 0,C 180,E1 -17169.418,E2 -17169.418} C_VEL
LIN {X 0,Y 287.629,Z 509.968,A -85,B 0,C 180,E1 -17171.885,E2 -17171.885} C_VEL
LIN {X 0,Y 286.014,Z 516.525,A -85,B 0,C 180,E1 -17174.319,E2 -17174.319} C_VEL
LIN {X 0,Y 284.444,Z 522.69,A -85,B 0,C 180,E1 -17177.152,E2 -17177.152} C_VEL
LIN {X 0,Y 283.484,Z 527.443,A -85,B 0,C 180,E1 -17180.006,E2 -17180.006} C_VEL
LIN {X 0,Y 282.891,Z 530.922,A -85,B 0,C 180,E1 -17182.865,E2 -17182.865} C_VEL
LIN {X 0,Y 282.545,Z 533.221,A -85,B 0,C 180,E1 -17185.721,E2 -17185.721} C_VEL
LIN {X 0,Y 282.371,Z 534.394,A -85,B 0,C 180,E1 -17188.574,E2 -17188.574} C_VEL
LIN {X 0,Y 282.371,Z 534.408,A -85,B 0,C 180,E1 -17191.426,E2 -17191.426} C_VEL
LIN {X 0,Y 282.538,Z 533.29,A -85,B 0,C 180,E1 -17194.279,E2 -17194.279} C_VEL
LIN {X 0,Y 282.834,Z 531.045,A -85,B 0,C 180,E1 -17197.137,E2 -17197.137} C_VEL
LIN {X 0,Y 283.468,Z 527.613,A -85,B 0,C 180,E1 -17199.994,E2 -17199.994} C_VEL
LIN {X 0,Y 284.419,Z 522.914,A -85,B 0,C 180,E1 -17202.849,E2 -17202.849} C_VEL
LIN {X 0,Y 285.992,Z 516.817,A -85,B 0,C 180,E1 -17205.683,E2 -17205.683} C_VEL
LIN {X 0,Y 287.903,Z 509.141,A -85,B 0,C 180,E1 -17208.502,E2 -17208.502} C_VEL
LIN {X 0,Y 290.145,Z 500.949,A -85,B 0,C 180,E1 -17210.933,E2 -17210.933} C_VEL
LIN {X 0,Y 292.798,Z 491.076,A -85,B 0,C 180,E1 -17213.331,E2 -17213.331} C_VEL
LIN {X 0,Y 295.289,Z 480.954,A -85,B 0,C 180,E1 -17215.366,E2 -17215.366} C_VEL
LIN {X 0,Y 298.304,Z 468.89,A -85,B 0,C 180,E1 -17217.349,E2 -17217.349} C_VEL
LIN {X 0,Y 300.885,Z 456.795,A -85,B 0,C 180,E1 -17218.99,E2 -17218.99} C_VEL
LIN {X 0,Y 303.522,Z 443.642,A -85,B 0,C 180,E1 -17220.431,E2 -17220.431} C_VEL
LIN {X 0,Y 305.699,Z 430.362,A -85,B 0,C 180,E1 -17221.607,E2 -17221.607} C_VEL
LIN {X 0,Y 307.564,Z 416.421,A -85,B 0,C 180,E1 -17222.575,E2 -17222.575} C_VEL
LIN {X 0,Y 309.132,Z 401.144,A -85,B 0,C 180,E1 -17223.359,E2 -17223.359} C_VEL
LIN {X 0,Y 310.274,Z 386.385,A -85,B 0,C 180,E1 -17223.853,E2 -17223.853} C_VEL
LIN {X 0,Y 313.342,Z 307.942,A -85,B 0,C 180,E1 -17225.639,E2 -17225.639} C_VEL
LIN {X 0,Y 314.295,Z 281.663,A -85,B 0,C 180,E1 -17226.241,E2 -17226.241} C_VEL
LIN {X 0,Y 306.263,Z 264.484,A -85,B 0,C 180,E1 -17227.857,E2 -17227.857} C_VEL
LIN {X 0,Y 298.471,Z 249.671,A -85,B 0,C 180,E1 -17229.489,E2 -17229.489} C_VEL
LIN {X 0,Y 293.444,Z 241.378,A -85,B 0,C 180,E1 -17230.569,E2 -17230.569} C_VEL
LIN {X 0,Y 288.958,Z 234.701,A -85,B 0,C 180,E1 -17231.558,E2 -17231.558} C_VEL
LIN {X 0,Y 288.721,Z 234.433,A -85,B 0,C 180,E1 -17231.608,E2 -17231.608} C_VEL
LIN {X 0,Y 287.275,Z 233.323,A -85,B 0,C 180,E1 -17231.903,E2 -17231.903} C_VEL
LIN {X 0,Y 284.352,Z 232.858,A -85,B 0,C 180,E1 -17232.453,E2 -17232.453} C_VEL
LIN {X 0,Y 280.42,Z 232.465,A -85,B 0,C 180,E1 -17233.21,E2 -17233.21} C_VEL
LIN {X 0,Y 279.613,Z 232.035,A -85,B 0,C 180,E1 -17233.382,E2 -17233.382} C_VEL
LIN {X 0,Y 277.934,Z 229.91,A -85,B 0,C 180,E1 -17233.786,E2 -17233.786} C_VEL
LIN {X 0,Y 277.22,Z 227.577,A -85,B 0,C 180,E1 -17234.047,E2 -17234.047} C_VEL
LIN {X 0,Y 277.216,Z 227.56,A -85,B 0,C 180,E1 -17237.323,E2 -17237.323} C_VEL
LIN {X 0,Y 277.277,Z 227.549,A -85,B 0,C 180,E1 -17241.788,E2 -17241.788} C_VEL
LIN {X 0,Y 277.3,Z 227.559,A -85,B 0,C 180,E1 -17244.344,E2 -17244.344} C_VEL
LIN {X 0,Y 277.24,Z 227.547,A -85,B 0,C 180,E1 -17247.836,E2 -17247.836} C_VEL
LIN {X 0,Y 277.285,Z 227.567,A -85,B 0,C 180,E1 -17251.212,E2 -17251.212} C_VEL
LIN {X 0,Y 277.309,Z 227.562,A -85,B 0,C 180,E1 -17254.479,E2 -17254.479} C_VEL
LIN {X 0,Y 277.28,Z 227.562,A -85,B 0,C 180,E1 -17257.654,E2 -17257.654} C_VEL
LIN {X 0,Y 277.339,Z 227.556,A -85,B 0,C 180,E1 -17260.766,E2 -17260.766} C_VEL
LIN {X 0,Y 277.422,Z 227.542,A -85,B 0,C 180,E1 -17265.325,E2 -17265.325} C_VEL
LIN {X 0,Y 277.501,Z 227.533,A -85,B 0,C 180,E1 -17269.788,E2 -17269.788} C_VEL
LIN {X 0,Y 277.643,Z 227.527,A -85,B 0,C 180,E1 -17272.729,E2 -17272.729} C_VEL
LIN {X 0,Y 277.816,Z 227.496,A -85,B 0,C 180,E1 -17278.55,E2 -17278.55} C_VEL
LIN {X 0,Y 277.816,Z 227.504,A -85,B 0,C 180,E1 -17281.449,E2 -17281.449} C_VEL
LIN {X 0,Y 277.634,Z 227.524,A -85,B 0,C 180,E1 -17287.271,E2 -17287.271} C_VEL
LIN {X 0,Y 277.455,Z 227.548,A -85,B 0,C 180,E1 -17290.213,E2 -17290.213} C_VEL
LIN {X 0,Y 277.422,Z 227.555,A -85,B 0,C 180,E1 -17294.675,E2 -17294.675} C_VEL
LIN {X 0,Y 277.339,Z 227.567,A -85,B 0,C 180,E1 -17299.234,E2 -17299.234} C_VEL
LIN {X 0,Y 277.314,Z 227.568,A -85,B 0,C 180,E1 -17304.171,E2 -17304.171} C_VEL
LIN {X 0,Y 277.321,Z 227.568,A -85,B 0,C 180,E1 -17307.506,E2 -17307.506} C_VEL
LIN {X 0,Y 277.267,Z 227.573,A -85,B 0,C 180,E1 -17310.482,E2 -17310.482} C_VEL
LIN {X 0,Y 277.243,Z 227.571,A -85,B 0,C 180,E1 -17313.896,E2 -17313.896} C_VEL
LIN {X 0,Y 277.269,Z 227.572,A -85,B 0,C 180,E1 -17317.469,E2 -17317.469} C_VEL
LIN {X 0,Y 277.205,Z 227.553,A -85,B 0,C 180,E1 -17321.237,E2 -17321.237} C_VEL
LIN {X 0,Y 277.196,Z 227.623,A -85,B 0,C 180,E1 -17322.876,E2 -17322.876} C_VEL
LIN {X 0,Y 280.309,Z 237.179,A -85,B 0,C 180,E1 -17326.578,E2 -17326.578} C_VEL
LIN {X 0,Y 282.962,Z 241.626,A -85,B 0,C 180,E1 -17327.231,E2 -17327.231} C_VEL
LIN {X 0,Y 291.408,Z 256.477,A -85,B 0,C 180,E1 -17329.214,E2 -17329.214} C_VEL
LIN {X 0,Y 299.21,Z 271.874,A -85,B 0,C 180,E1 -17330.949,E2 -17330.949} C_VEL
LIN {X 0,Y 306.727,Z 288.892,A -85,B 0,C 180,E1 -17332.564,E2 -17332.564} C_VEL
LIN {X 0,Y 307.436,Z 291.257,A -85,B 0,C 180,E1 -17332.733,E2 -17332.733} C_VEL
LIN {X 0,Y 308.183,Z 296.669,A -85,B 0,C 180,E1 -17332.992,E2 -17332.992} C_VEL
LIN {X 0,Y 303.699,Z 403.888,A -85,B 0,C 180,E1 -17335.462,E2 -17335.462} C_VEL
LIN {X 0,Y 302.281,Z 420.109,A -85,B 0,C 180,E1 -17336.084,E2 -17336.084} C_VEL
LIN {X 0,Y 300.213,Z 435.382,A -85,B 0,C 180,E1 -17336.925,E2 -17336.925} C_VEL
LIN {X 0,Y 298.036,Z 449.141,A -85,B 0,C 180,E1 -17337.957,E2 -17337.957} C_VEL
LIN {X 0,Y 295.48,Z 462.608,A -85,B 0,C 180,E1 -17339.245,E2 -17339.245} C_VEL
LIN {X 0,Y 292.409,Z 476.33,A -85,B 0,C 180,E1 -17340.877,E2 -17340.877} C_VEL
LIN {X 0,Y 289.356,Z 488.758,A -85,B 0,C 180,E1 -17342.714,E2 -17342.714} C_VEL
LIN {X 0,Y 286.175,Z 500.949,A -85,B 0,C 180,E1 -17344.937,E2 -17344.937} C_VEL
LIN {X 0,Y 283.727,Z 510.362,A -85,B 0,C 180,E1 -17347.038,E2 -17347.038} C_VEL
LIN {X 0,Y 281.113,Z 519.622,A -85,B 0,C 180,E1 -17349.513,E2 -17349.513} C_VEL
LIN {X 0,Y 278.856,Z 528.348,A -85,B 0,C 180,E1 -17352.397,E2 -17352.397} C_VEL
LIN {X 0,Y 277.232,Z 535.358,A -85,B 0,C 180,E1 -17355.315,E2 -17355.315} C_VEL
LIN {X 0,Y 276.073,Z 540.872,A -85,B 0,C 180,E1 -17358.249,E2 -17358.249} C_VEL
LIN {X 0,Y 275.473,Z 545.049,A -85,B 0,C 180,E1 -17361.195,E2 -17361.195} C_VEL
LIN {X 0,Y 275.233,Z 547.98,A -85,B 0,C 180,E1 -17364.138,E2 -17364.138} C_VEL
LIN {X 0,Y 275.231,Z 549.73,A -85,B 0,C 180,E1 -17367.073,E2 -17367.073} C_VEL
LIN {X 0,Y 275.276,Z 550.329,A -85,B 0,C 180,E1 -17370,E2 -17370} C_VEL
LIN {X 0,Y 275.231,Z 549.719,A -85,B 0,C 180,E1 -17372.927,E2 -17372.927} C_VEL
LIN {X 0,Y 275.233,Z 547.954,A -85,B 0,C 180,E1 -17375.862,E2 -17375.862} C_VEL
LIN {X 0,Y 275.473,Z 545.013,A -85,B 0,C 180,E1 -17378.805,E2 -17378.805} C_VEL
LIN {X 0,Y 276.071,Z 540.83,A -85,B 0,C 180,E1 -17381.751,E2 -17381.751} C_VEL
LIN {X 0,Y 277.207,Z 535.297,A -85,B 0,C 180,E1 -17384.686,E2 -17384.686} C_VEL
LIN {X 0,Y 278.384,Z 530.152,A -85,B 0,C 180,E1 -17386.877,E2 -17386.877} C_VEL
LIN {X 0,Y 280.208,Z 523,A -85,B 0,C 180,E1 -17389.41,E2 -17389.41} C_VEL
LIN {X 0,Y 282.592,Z 514.419,A -85,B 0,C 180,E1 -17391.903,E2 -17391.903} C_VEL
LIN {X 0,Y 284.92,Z 505.267,A -85,B 0,C 180,E1 -17394.125,E2 -17394.125} C_VEL
LIN {X 0,Y 287.569,Z 495.459,A -85,B 0,C 180,E1 -17396.097,E2 -17396.097} C_VEL
LIN {X 0,Y 290.681,Z 483.223,A -85,B 0,C 180,E1 -17398.129,E2 -17398.129} C_VEL
LIN {X 0,Y 293.889,Z 469.6,A -85,B 0,C 180,E1 -17399.946,E2 -17399.946} C_VEL
LIN {X 0,Y 296.711,Z 455.943,A -85,B 0,C 180,E1 -17401.405,E2 -17401.405} C_VEL
LIN {X 0,Y 299.195,Z 441.795,A -85,B 0,C 180,E1 -17402.601,E2 -17402.601} C_VEL
LIN {X 0,Y 301.289,Z 427.224,A -85,B 0,C 180,E1 -17403.541,E2 -17403.541} C_VEL
LIN {X 0,Y 302.976,Z 412.264,A -85,B 0,C 180,E1 -17404.229,E2 -17404.229} C_VEL
LIN {X 0,Y 304.034,Z 396.859,A -85,B 0,C 180,E1 -17404.695,E2 -17404.695} C_VEL
LIN {X 0,Y 308.089,Z 296.945,A -85,B 0,C 180,E1 -17406.978,E2 -17406.978} C_VEL
LIN {X 0,Y 306.907,Z 289.403,A -85,B 0,C 180,E1 -17407.36,E2 -17407.36} C_VEL
LIN {X 0,Y 298.827,Z 271.083,A -85,B 0,C 180,E1 -17409.094,E2 -17409.094} C_VEL
LIN {X 0,Y 290.874,Z 255.516,A -85,B 0,C 180,E1 -17410.863,E2 -17410.863} C_VEL
LIN {X 0,Y 284.863,Z 245.038,A -85,B 0,C 180,E1 -17412.256,E2 -17412.256} C_VEL
LIN {X 0,Y 282.247,Z 240.641,A -85,B 0,C 180,E1 -17412.886,E2 -17412.886} C_VEL
LIN {X 0,Y 280.15,Z 236.831,A -85,B 0,C 180,E1 -17413.453,E2 -17413.453} C_VEL
LIN {X 0,Y 277.2,Z 227.574,A -85,B 0,C 180,E1 -17417.122,E2 -17417.122} C_VEL
LIN {X 0,Y 277.262,Z 227.569,A -85,B 0,C 180,E1 -17420.677,E2 -17420.677} C_VEL
LIN {X 0,Y 277.3,Z 227.557,A -85,B 0,C 180,E1 -17424.344,E2 -17424.344} C_VEL
LIN {X 0,Y 277.242,Z 227.567,A -85,B 0,C 180,E1 -17427.836,E2 -17427.836} C_VEL
LIN {X 0,Y 277.3,Z 227.564,A -85,B 0,C 180,E1 -17431.214,E2 -17431.214} C_VEL
LIN {X 0,Y 277.304,Z 227.568,A -85,B 0,C 180,E1 -17434.479,E2 -17434.479} C_VEL
LIN {X 0,Y 277.261,Z 227.542,A -85,B 0,C 180,E1 -17437.653,E2 -17437.653} C_VEL
LIN {X 0,Y 277.339,Z 227.559,A -85,B 0,C 180,E1 -17440.766,E2 -17440.766} C_VEL
LIN {X 0,Y 277.422,Z 227.553,A -85,B 0,C 180,E1 -17445.325,E2 -17445.325} C_VEL
LIN {X 0,Y 277.455,Z 227.549,A -85,B 0,C 180,E1 -17449.787,E2 -17449.787} C_VEL
LIN {X 0,Y 277.634,Z 227.523,A -85,B 0,C 180,E1 -17452.729,E2 -17452.729} C_VEL
LIN {X 0,Y 277.816,Z 227.503,A -85,B 0,C 180,E1 -17458.551,E2 -17458.551} C_VEL
LIN {X 0,Y 277.816,Z 227.501,A -85,B 0,C 180,E1 -17461.45,E2 -17461.45} C_VEL
LIN {X 0,Y 277.635,Z 227.524,A -85,B 0,C 180,E1 -17467.272,E2 -17467.272} C_VEL
LIN {X 0,Y 277.455,Z 227.548,A -85,B 0,C 180,E1 -17470.213,E2 -17470.213} C_VEL
LIN {X 0,Y 277.422,Z 227.553,A -85,B 0,C 180,E1 -17474.675,E2 -17474.675} C_VEL
LIN {X 0,Y 277.337,Z 227.563,A -85,B 0,C 180,E1 -17479.235,E2 -17479.235} C_VEL
LIN {X 0,Y 277.286,Z 227.555,A -85,B 0,C 180,E1 -17484.158,E2 -17484.158} C_VEL
LIN {X 0,Y 277.32,Z 227.543,A -85,B 0,C 180,E1 -17487.505,E2 -17487.505} C_VEL
LIN {X 0,Y 277.268,Z 227.568,A -85,B 0,C 180,E1 -17490.482,E2 -17490.482} C_VEL
LIN {X 0,Y 277.243,Z 227.568,A -85,B 0,C 180,E1 -17493.896,E2 -17493.896} C_VEL
LIN {X 0,Y 277.264,Z 227.567,A -85,B 0,C 180,E1 -17497.47,E2 -17497.47} C_VEL
LIN {X 0,Y 277.206,Z 227.574,A -85,B 0,C 180,E1 -17501.237,E2 -17501.237} C_VEL
LIN {X 0,Y 277.214,Z 227.579,A -85,B 0,C 180,E1 -17505.224,E2 -17505.224} C_VEL
LIN {X 0,Y 277.227,Z 227.626,A -85,B 0,C 180,E1 -17506.135,E2 -17506.135} C_VEL
LIN {X 0,Y 278.217,Z 230.375,A -85,B 0,C 180,E1 -17506.429,E2 -17506.429} C_VEL
LIN {X 0,Y 280.412,Z 233.11,A -85,B 0,C 180,E1 -17506.952,E2 -17506.952} C_VEL
LIN {X 0,Y 282.694,Z 236.49,A -85,B 0,C 180,E1 -17507.5,E2 -17507.5} C_VEL
LIN {X 0,Y 291.467,Z 249.831,A -85,B 0,C 180,E1 -17509.499,E2 -17509.499} C_VEL
LIN {X 0,Y 299.452,Z 264.677,A -85,B 0,C 180,E1 -17511.252,E2 -17511.252} C_VEL
LIN {X 0,Y 307.592,Z 281.943,A -85,B 0,C 180,E1 -17512.966,E2 -17512.966} C_VEL
LIN {X 0,Y 308.487,Z 284.006,A -85,B 0,C 180,E1 -17513.151,E2 -17513.151} C_VEL
LIN {X 0,Y 304.189,Z 388.867,A -85,B 0,C 180,E1 -17515.576,E2 -17515.576} C_VEL
LIN {X 0,Y 302.908,Z 404.569,A -85,B 0,C 180,E1 -17516.163,E2 -17516.163} C_VEL
LIN {X 0,Y 301.185,Z 419.688,A -85,B 0,C 180,E1 -17517.006,E2 -17517.006} C_VEL
LIN {X 0,Y 299.383,Z 432.176,A -85,B 0,C 180,E1 -17517.933,E2 -17517.933} C_VEL
LIN {X 0,Y 296.934,Z 446.002,A -85,B 0,C 180,E1 -17519.215,E2 -17519.215} C_VEL
LIN {X 0,Y 294.273,Z 458.766,A -85,B 0,C 180,E1 -17520.687,E2 -17520.687} C_VEL
LIN {X 0,Y 291.228,Z 471.624,A -85,B 0,C 180,E1 -17522.515,E2 -17522.515} C_VEL
LIN {X 0,Y 288.203,Z 483.614,A -85,B 0,C 180,E1 -17524.625,E2 -17524.625} C_VEL
LIN {X 0,Y 285.46,Z 493.774,A -85,B 0,C 180,E1 -17526.802,E2 -17526.802} C_VEL
LIN {X 0,Y 282.875,Z 503.213,A -85,B 0,C 180,E1 -17529.266,E2 -17529.266} C_VEL
LIN {X 0,Y 280.324,Z 512.07,A -85,B 0,C 180,E1 -17532.115,E2 -17532.115} C_VEL
LIN {X 0,Y 278.725,Z 518.396,A -85,B 0,C 180,E1 -17534.648,E2 -17534.648} C_VEL
LIN {X 0,Y 277.194,Z 524.209,A -85,B 0,C 180,E1 -17537.555,E2 -17537.555} C_VEL
LIN {X 0,Y 276.464,Z 527.646,A -85,B 0,C 180,E1 -17539.75,E2 -17539.75} C_VEL
LIN {X 0,Y 275.821,Z 531.125,A -85,B 0,C 180,E1 -17542.681,E2 -17542.681} C_VEL
LIN {X 0,Y 275.471,Z 533.422,A -85,B 0,C 180,E1 -17545.61,E2 -17545.61} C_VEL
LIN {X 0,Y 275.297,Z 534.595,A -85,B 0,C 180,E1 -17548.537,E2 -17548.537} C_VEL
LIN {X 0,Y 275.297,Z 534.608,A -85,B 0,C 180,E1 -17551.463,E2 -17551.463} C_VEL
LIN {X 0,Y 275.445,Z 533.491,A -85,B 0,C 180,E1 -17554.39,E2 -17554.39} C_VEL
LIN {X 0,Y 275.777,Z 531.246,A -85,B 0,C 180,E1 -17557.32,E2 -17557.32} C_VEL
LIN {X 0,Y 276.448,Z 527.814,A -85,B 0,C 180,E1 -17560.251,E2 -17560.251} C_VEL
LIN {X 0,Y 277.467,Z 523.115,A -85,B 0,C 180,E1 -17563.177,E2 -17563.177} C_VEL
LIN {X 0,Y 279.098,Z 517.018,A -85,B 0,C 180,E1 -17566.08,E2 -17566.08} C_VEL
LIN {X 0,Y 281.132,Z 509.341,A -85,B 0,C 180,E1 -17568.964,E2 -17568.964} C_VEL
LIN {X 0,Y 283.486,Z 501.148,A -85,B 0,C 180,E1 -17571.448,E2 -17571.448} C_VEL
LIN {X 0,Y 286.282,Z 491.274,A -85,B 0,C 180,E1 -17573.894,E2 -17573.894} C_VEL
LIN {X 0,Y 288.887,Z 481.152,A -85,B 0,C 180,E1 -17575.969,E2 -17575.969} C_VEL
LIN {X 0,Y 291.732,Z 470.153,A -85,B 0,C 180,E1 -17577.823,E2 -17577.823} C_VEL
LIN {X 0,Y 294.396,Z 458.278,A -85,B 0,C 180,E1 -17579.496,E2 -17579.496} C_VEL
LIN {X 0,Y 297.129,Z 445.413,A -85,B 0,C 180,E1 -17580.96,E2 -17580.96} C_VEL
LIN {X 0,Y 299.546,Z 431.362,A -85,B 0,C 180,E1 -17582.253,E2 -17582.253} C_VEL
LIN {X 0,Y 301.622,Z 416.613,A -85,B 0,C 180,E1 -17583.299,E2 -17583.299} C_VEL
LIN {X 0,Y 303.248,Z 401.332,A -85,B 0,C 180,E1 -17584.094,E2 -17584.094} C_VEL
LIN {X 0,Y 304.415,Z 386.565,A -85,B 0,C 180,E1 -17584.596,E2 -17584.596} C_VEL
LIN {X 0,Y 307.605,Z 307.84,A -85,B 0,C 180,E1 -17586.417,E2 -17586.417} C_VEL
LIN {X 0,Y 308.491,Z 283.837,A -85,B 0,C 180,E1 -17586.978,E2 -17586.978} C_VEL
LIN {X 0,Y 301.282,Z 268.348,A -85,B 0,C 180,E1 -17588.486,E2 -17588.486} C_VEL
LIN {X 0,Y 294.046,Z 254.384,A -85,B 0,C 180,E1 -17590.06,E2 -17590.06} C_VEL
LIN {X 0,Y 289.395,Z 246.598,A -85,B 0,C 180,E1 -17591.095,E2 -17591.095} C_VEL
LIN {X 0,Y 282.419,Z 236.17,A -85,B 0,C 180,E1 -17592.702,E2 -17592.702} C_VEL
LIN {X 0,Y 280.293,Z 232.848,A -85,B 0,C 180,E1 -17593.222,E2 -17593.222} C_VEL
LIN {X 0,Y 279.613,Z 232.035,A -85,B 0,C 180,E1 -17593.382,E2 -17593.382} C_VEL
LIN {X 0,Y 276.333,Z 230.032,A -85,B 0,C 180,E1 -17594.295,E2 -17594.295} C_VEL
LIN {X 0,Y 273.774,Z 228.927,A -85,B 0,C 180,E1 -17595.38,E2 -17595.38} C_VEL
LIN {X 0,Y 271.473,Z 228.41,A -85,B 0,C 180,E1 -17596.987,E2 -17596.987} C_VEL
LIN {X 0,Y 270.333,Z 228.428,A -85,B 0,C 180,E1 -17598.687,E2 -17598.687} C_VEL
LIN {X 0,Y 270.169,Z 228.452,A -85,B 0,C 180,E1 -17599.548,E2 -17599.548} C_VEL
LIN {X 0,Y 270.252,Z 228.427,A -85,B 0,C 180,E1 -17603.721,E2 -17603.721} C_VEL
LIN {X 0,Y 270.2,Z 228.435,A -85,B 0,C 180,E1 -17606.892,E2 -17606.892} C_VEL
LIN {X 0,Y 270.225,Z 228.434,A -85,B 0,C 180,E1 -17610.386,E2 -17610.386} C_VEL
LIN {X 0,Y 270.259,Z 228.437,A -85,B 0,C 180,E1 -17613.763,E2 -17613.763} C_VEL
LIN {X 0,Y 270.227,Z 228.441,A -85,B 0,C 180,E1 -17617.038,E2 -17617.038} C_VEL
LIN {X 0,Y 270.296,Z 228.439,A -85,B 0,C 180,E1 -17620.244,E2 -17620.244} C_VEL
LIN {X 0,Y 270.391,Z 228.42,A -85,B 0,C 180,E1 -17624.935,E2 -17624.935} C_VEL
LIN {X 0,Y 270.436,Z 228.414,A -85,B 0,C 180,E1 -17629.519,E2 -17629.519} C_VEL
LIN {X 0,Y 270.602,Z 228.404,A -85,B 0,C 180,E1 -17632.538,E2 -17632.538} C_VEL
LIN {X 0,Y 270.782,Z 228.372,A -85,B 0,C 180,E1 -17638.513,E2 -17638.513} C_VEL
LIN {X 0,Y 270.782,Z 228.38,A -85,B 0,C 180,E1 -17641.487,E2 -17641.487} C_VEL
LIN {X 0,Y 270.592,Z 228.4,A -85,B 0,C 180,E1 -17647.462,E2 -17647.462} C_VEL
LIN {X 0,Y 270.407,Z 228.429,A -85,B 0,C 180,E1 -17650.482,E2 -17650.482} C_VEL
LIN {X 0,Y 270.391,Z 228.433,A -85,B 0,C 180,E1 -17655.065,E2 -17655.065} C_VEL
LIN {X 0,Y 270.296,Z 228.445,A -85,B 0,C 180,E1 -17659.756,E2 -17659.756} C_VEL
LIN {X 0,Y 270.269,Z 228.441,A -85,B 0,C 180,E1 -17664.586,E2 -17664.586} C_VEL
LIN {X 0,Y 270.267,Z 228.447,A -85,B 0,C 180,E1 -17667.909,E2 -17667.909} C_VEL
LIN {X 0,Y 270.18,Z 228.456,A -85,B 0,C 180,E1 -17671.349,E2 -17671.349} C_VEL
LIN {X 0,Y 270.198,Z 228.453,A -85,B 0,C 180,E1 -17674.906,E2 -17674.906} C_VEL
LIN {X 0,Y 270.193,Z 228.441,A -85,B 0,C 180,E1 -17678.711,E2 -17678.711} C_VEL
LIN {X 0,Y 270.169,Z 228.534,A -85,B 0,C 180,E1 -17681.674,E2 -17681.674} C_VEL
LIN {X 0,Y 272.863,Z 236.905,A -85,B 0,C 180,E1 -17685.079,E2 -17685.079} C_VEL
LIN {X 0,Y 275.86,Z 241.688,A -85,B 0,C 180,E1 -17685.862,E2 -17685.862} C_VEL
LIN {X 0,Y 282.302,Z 252.64,A -85,B 0,C 180,E1 -17687.48,E2 -17687.48} C_VEL
LIN {X 0,Y 290.147,Z 267.264,A -85,B 0,C 180,E1 -17689.345,E2 -17689.345} C_VEL
LIN {X 0,Y 296.874,Z 281.358,A -85,B 0,C 180,E1 -17690.875,E2 -17690.875} C_VEL
LIN {X 0,Y 301.878,Z 293.279,A -85,B 0,C 180,E1 -17691.991,E2 -17691.991} C_VEL
LIN {X 0,Y 302.485,Z 298.256,A -85,B 0,C 180,E1 -17692.226,E2 -17692.226} C_VEL
LIN {X 0,Y 297.89,Z 403.704,A -85,B 0,C 180,E1 -17694.69,E2 -17694.69} C_VEL
LIN {X 0,Y 296.511,Z 419.092,A -85,B 0,C 180,E1 -17695.279,E2 -17695.279} C_VEL
LIN {X 0,Y 294.455,Z 433.982,A -85,B 0,C 180,E1 -17696.09,E2 -17696.09} C_VEL
LIN {X 0,Y 292.025,Z 448.946,A -85,B 0,C 180,E1 -17697.216,E2 -17697.216} C_VEL
LIN {X 0,Y 289.296,Z 462.851,A -85,B 0,C 180,E1 -17698.57,E2 -17698.57} C_VEL
LIN {X 0,Y 286.203,Z 476.132,A -85,B 0,C 180,E1 -17700.182,E2 -17700.182} C_VEL
LIN {X 0,Y 283.027,Z 488.559,A -85,B 0,C 180,E1 -17702.051,E2 -17702.051} C_VEL
LIN {X 0,Y 279.693,Z 500.749,A -85,B 0,C 180,E1 -17704.314,E2 -17704.314} C_VEL
LIN {X 0,Y 277.117,Z 510.161,A -85,B 0,C 180,E1 -17706.458,E2 -17706.458} C_VEL
LIN {X 0,Y 274.409,Z 519.421,A -85,B 0,C 180,E1 -17708.989,E2 -17708.989} C_VEL
LIN {X 0,Y 272.022,Z 528.146,A -85,B 0,C 180,E1 -17711.939,E2 -17711.939} C_VEL
LIN {X 0,Y 270.311,Z 535.156,A -85,B 0,C 180,E1 -17714.93,E2 -17714.93} C_VEL
LIN {X 0,Y 269.072,Z 540.671,A -85,B 0,C 180,E1 -17717.939,E2 -17717.939} C_VEL
LIN {X 0,Y 268.414,Z 544.847,A -85,B 0,C 180,E1 -17720.962,E2 -17720.962} C_VEL
LIN {X 0,Y 268.144,Z 547.779,A -85,B 0,C 180,E1 -17723.982,E2 -17723.982} C_VEL
LIN {X 0,Y 268.143,Z 549.529,A -85,B 0,C 180,E1 -17726.995,E2 -17726.995} C_VEL
LIN {X 0,Y 268.2,Z 550.129,A -85,B 0,C 180,E1 -17730,E2 -17730} C_VEL
LIN {X 0,Y 268.143,Z 549.518,A -85,B 0,C 180,E1 -17733.005,E2 -17733.005} C_VEL
LIN {X 0,Y 268.144,Z 547.752,A -85,B 0,C 180,E1 -17736.018,E2 -17736.018} C_VEL
LIN {X 0,Y 268.414,Z 544.81,A -85,B 0,C 180,E1 -17739.038,E2 -17739.038} C_VEL
LIN {X 0,Y 269.07,Z 540.626,A -85,B 0,C 180,E1 -17742.061,E2 -17742.061} C_VEL
LIN {X 0,Y 270.27,Z 535.092,A -85,B 0,C 180,E1 -17745.072,E2 -17745.072} C_VEL
LIN {X 0,Y 272.022,Z 528.06,A -85,B 0,C 180,E1 -17748.061,E2 -17748.061} C_VEL
LIN {X 0,Y 274.414,Z 519.318,A -85,B 0,C 180,E1 -17751.011,E2 -17751.011} C_VEL
LIN {X 0,Y 277.103,Z 510.04,A -85,B 0,C 180,E1 -17753.544,E2 -17753.544} C_VEL
LIN {X 0,Y 279.718,Z 500.611,A -85,B 0,C 180,E1 -17755.684,E2 -17755.684} C_VEL
LIN {X 0,Y 282.983,Z 488.385,A -85,B 0,C 180,E1 -17757.954,E2 -17757.954} C_VEL
LIN {X 0,Y 286.197,Z 475.924,A -85,B 0,C 180,E1 -17759.819,E2 -17759.819} C_VEL
LIN {X 0,Y 289.242,Z 462.659,A -85,B 0,C 180,E1 -17761.426,E2 -17761.426} C_VEL
LIN {X 0,Y 292.007,Z 448.601,A -85,B 0,C 180,E1 -17762.786,E2 -17762.786} C_VEL
LIN {X 0,Y 294.416,Z 433.543,A -85,B 0,C 180,E1 -17763.916,E2 -17763.916} C_VEL
LIN {X 0,Y 296.429,Z 418.476,A -85,B 0,C 180,E1 -17764.732,E2 -17764.732} C_VEL
LIN {X 0,Y 297.893,Z 402.67,A -85,B 0,C 180,E1 -17765.31,E2 -17765.31} C_VEL
LIN {X 0,Y 302.417,Z 297.884,A -85,B 0,C 180,E1 -17767.757,E2 -17767.757} C_VEL
LIN {X 0,Y 301.512,Z 292.257,A -85,B 0,C 180,E1 -17768.056,E2 -17768.056} C_VEL
LIN {X 0,Y 293.314,Z 273.694,A -85,B 0,C 180,E1 -17769.886,E2 -17769.886} C_VEL
LIN {X 0,Y 285.691,Z 258.81,A -85,B 0,C 180,E1 -17771.653,E2 -17771.653} C_VEL
LIN {X 0,Y 278.475,Z 246.048,A -85,B 0,C 180,E1 -17773.418,E2 -17773.418} C_VEL
LIN {X 0,Y 272.716,Z 236.527,A -85,B 0,C 180,E1 -17774.957,E2 -17774.957} C_VEL
LIN {X 0,Y 270.188,Z 228.451,A -85,B 0,C 180,E1 -17778.374,E2 -17778.374} C_VEL
LIN {X 0,Y 270.241,Z 228.438,A -85,B 0,C 180,E1 -17781.38,E2 -17781.38} C_VEL
LIN {X 0,Y 270.211,Z 228.442,A -85,B 0,C 180,E1 -17785.096,E2 -17785.096} C_VEL
LIN {X 0,Y 270.196,Z 228.449,A -85,B 0,C 180,E1 -17789.13,E2 -17789.13} C_VEL
LIN {X 0,Y 270.263,Z 228.441,A -85,B 0,C 180,E1 -17792.144,E2 -17792.144} C_VEL
LIN {X 0,Y 270.233,Z 228.446,A -85,B 0,C 180,E1 -17795.537,E2 -17795.537} C_VEL
LIN {X 0,Y 270.296,Z 228.425,A -85,B 0,C 180,E1 -17800.244,E2 -17800.244} C_VEL
LIN {X 0,Y 270.391,Z 228.427,A -85,B 0,C 180,E1 -17804.935,E2 -17804.935} C_VEL
LIN {X 0,Y 270.407,Z 228.429,A -85,B 0,C 180,E1 -17809.518,E2 -17809.518} C_VEL
LIN {X 0,Y 270.592,Z 228.399,A -85,B 0,C 180,E1 -17812.538,E2 -17812.538} C_VEL
LIN {X 0,Y 270.782,Z 228.38,A -85,B 0,C 180,E1 -17818.513,E2 -17818.513} C_VEL
LIN {X 0,Y 270.782,Z 228.378,A -85,B 0,C 180,E1 -17821.487,E2 -17821.487} C_VEL
LIN {X 0,Y 270.593,Z 228.399,A -85,B 0,C 180,E1 -17827.462,E2 -17827.462} C_VEL
LIN {X 0,Y 270.407,Z 228.426,A -85,B 0,C 180,E1 -17830.483,E2 -17830.483} C_VEL
LIN {X 0,Y 270.391,Z 228.431,A -85,B 0,C 180,E1 -17835.065,E2 -17835.065} C_VEL
LIN {X 0,Y 270.295,Z 228.437,A -85,B 0,C 180,E1 -17839.756,E2 -17839.756} C_VEL
LIN {X 0,Y 270.233,Z 228.425,A -85,B 0,C 180,E1 -17844.59,E2 -17844.59} C_VEL
LIN {X 0,Y 270.268,Z 228.427,A -85,B 0,C 180,E1 -17847.909,E2 -17847.909} C_VEL
LIN {X 0,Y 270.18,Z 228.45,A -85,B 0,C 180,E1 -17851.349,E2 -17851.349} C_VEL
LIN {X 0,Y 270.198,Z 228.449,A -85,B 0,C 180,E1 -17854.906,E2 -17854.906} C_VEL
LIN {X 0,Y 270.194,Z 228.448,A -85,B 0,C 180,E1 -17858.711,E2 -17858.711} C_VEL
LIN {X 0,Y 270.169,Z 228.455,A -85,B 0,C 180,E1 -17863.251,E2 -17863.251} C_VEL
LIN {X 0,Y 270.168,Z 228.452,A -85,B 0,C 180,E1 -17864.698,E2 -17864.698} C_VEL
LIN {X 0,Y 271.074,Z 231.132,A -85,B 0,C 180,E1 -17864.991,E2 -17864.991} C_VEL
LIN {X 0,Y 273.511,Z 234.07,A -85,B 0,C 180,E1 -17865.61,E2 -17865.61} C_VEL
LIN {X 0,Y 275.526,Z 237.176,A -85,B 0,C 180,E1 -17866.132,E2 -17866.132} C_VEL
LIN {X 0,Y 277.012,Z 239.347,A -85,B 0,C 180,E1 -17866.506,E2 -17866.506} C_VEL
LIN {X 0,Y 284.239,Z 249.985,A -85,B 0,C 180,E1 -17868.238,E2 -17868.238} C_VEL
LIN {X 0,Y 289.99,Z 259.728,A -85,B 0,C 180,E1 -17869.565,E2 -17869.565} C_VEL
LIN {X 0,Y 298.346,Z 276.351,A -85,B 0,C 180,E1 -17871.434,E2 -17871.434} C_VEL
LIN {X 0,Y 302.751,Z 286.122,A -85,B 0,C 180,E1 -17872.389,E2 -17872.389} C_VEL
LIN {X 0,Y 298.46,Z 387.583,A -85,B 0,C 180,E1 -17874.767,E2 -17874.767} C_VEL
LIN {X 0,Y 297.304,Z 402.039,A -85,B 0,C 180,E1 -17875.282,E2 -17875.282} C_VEL
LIN {X 0,Y 295.661,Z 416.526,A -85,B 0,C 180,E1 -17876.041,E2 -17876.041} C_VEL
LIN {X 0,Y 293.416,Z 431.807,A -85,B 0,C 180,E1 -17877.14,E2 -17877.14} C_VEL
LIN {X 0,Y 291.168,Z 444.631,A -85,B 0,C 180,E1 -17878.334,E2 -17878.334} C_VEL
LIN {X 0,Y 288.412,Z 457.684,A -85,B 0,C 180,E1 -17879.829,E2 -17879.829} C_VEL
LIN {X 0,Y 285.536,Z 469.7,A -85,B 0,C 180,E1 -17881.519,E2 -17881.519} C_VEL
LIN {X 0,Y 282.595,Z 480.798,A -85,B 0,C 180,E1 -17883.408,E2 -17883.408} C_VEL
LIN {X 0,Y 279.881,Z 490.974,A -85,B 0,C 180,E1 -17885.524,E2 -17885.524} C_VEL
LIN {X 0,Y 276.938,Z 500.932,A -85,B 0,C 180,E1 -17888.018,E2 -17888.018} C_VEL
LIN {X 0,Y 274.466,Z 509.186,A -85,B 0,C 180,E1 -17890.557,E2 -17890.557} C_VEL
LIN {X 0,Y 272.515,Z 515.818,A -85,B 0,C 180,E1 -17893.04,E2 -17893.04} C_VEL
LIN {X 0,Y 270.973,Z 521.685,A -85,B 0,C 180,E1 -17895.736,E2 -17895.736} C_VEL
LIN {X 0,Y 269.68,Z 526.797,A -85,B 0,C 180,E1 -17898.729,E2 -17898.729} C_VEL
LIN {X 0,Y 269.051,Z 529.74,A -85,B 0,C 180,E1 -17900.983,E2 -17900.983} C_VEL
LIN {X 0,Y 268.493,Z 532.691,A -85,B 0,C 180,E1 -17904.087,E2 -17904.087} C_VEL
LIN {X 0,Y 268.306,Z 534.347,A -85,B 0,C 180,E1 -17906.997,E2 -17906.997} C_VEL
LIN {X 0,Y 268.207,Z 534.951,A -85,B 0,C 180,E1 -17910,E2 -17910} C_VEL
LIN {X 0,Y 268.303,Z 534.388,A -85,B 0,C 180,E1 -17913.003,E2 -17913.003} C_VEL
LIN {X 0,Y 268.505,Z 532.713,A -85,B 0,C 180,E1 -17916.01,E2 -17916.01} C_VEL
LIN {X 0,Y 269.022,Z 529.883,A -85,B 0,C 180,E1 -17919.018,E2 -17919.018} C_VEL
LIN {X 0,Y 269.935,Z 525.83,A -85,B 0,C 180,E1 -17922.022,E2 -17922.022} C_VEL
LIN {X 0,Y 271.387,Z 520.449,A -85,B 0,C 180,E1 -17925.008,E2 -17925.008} C_VEL
LIN {X 0,Y 273.248,Z 513.593,A -85,B 0,C 180,E1 -17927.977,E2 -17927.977} C_VEL
LIN {X 0,Y 275.423,Z 506.215,A -85,B 0,C 180,E1 -17930.539,E2 -17930.539} C_VEL
LIN {X 0,Y 278.021,Z 497.32,A -85,B 0,C 180,E1 -17933.067,E2 -17933.067} C_VEL
LIN {X 0,Y 280.684,Z 488.243,A -85,B 0,C 180,E1 -17935.192,E2 -17935.192} C_VEL
LIN {X 0,Y 283.023,Z 479.479,A -85,B 0,C 180,E1 -17936.947,E2 -17936.947} C_VEL
LIN {X 0,Y 286.018,Z 468.176,A -85,B 0,C 180,E1 -17938.83,E2 -17938.83} C_VEL
LIN {X 0,Y 288.525,Z 457.189,A -85,B 0,C 180,E1 -17940.36,E2 -17940.36} C_VEL
LIN {X 0,Y 291.373,Z 444.033,A -85,B 0,C 180,E1 -17941.845,E2 -17941.845} C_VEL
LIN {X 0,Y 293.778,Z 430.322,A -85,B 0,C 180,E1 -17943.093,E2 -17943.093} C_VEL
LIN {X 0,Y 295.889,Z 415.507,A -85,B 0,C 180,E1 -17944.134,E2 -17944.134} C_VEL
LIN {X 0,Y 297.409,Z 401.52,A -85,B 0,C 180,E1 -17944.859,E2 -17944.859} C_VEL
LIN {X 0,Y 298.607,Z 386.745,A -85,B 0,C 180,E1 -17945.368,E2 -17945.368} C_VEL
LIN {X 0,Y 301.918,Z 308.216,A -85,B 0,C 180,E1 -17947.211,E2 -17947.211} C_VEL
LIN {X 0,Y 302.858,Z 286.347,A -85,B 0,C 180,E1 -17947.716,E2 -17947.716} C_VEL
LIN {X 0,Y 296.01,Z 271.455,A -85,B 0,C 180,E1 -17949.212,E2 -17949.212} C_VEL
LIN {X 0,Y 289.02,Z 257.922,A -85,B 0,C 180,E1 -17950.794,E2 -17950.794} C_VEL
LIN {X 0,Y 283.766,Z 249.237,A -85,B 0,C 180,E1 -17952.012,E2 -17952.012} C_VEL
LIN {X 0,Y 278.069,Z 240.877,A -85,B 0,C 180,E1 -17953.376,E2 -17953.376} C_VEL
LIN {X 0,Y 275.539,Z 237.187,A -85,B 0,C 180,E1 -17954.009,E2 -17954.009} C_VEL
LIN {X 0,Y 273.416,Z 233.894,A -85,B 0,C 180,E1 -17954.562,E2 -17954.562} C_VEL
LIN {X 0,Y 270.883,Z 230.791,A -85,B 0,C 180,E1 -17955.21,E2 -17955.21} C_VEL
LIN {X 0,Y 270.176,Z 228.457,A -85,B 0,C 180,E1 -17955.479,E2 -17955.479} C_VEL
LIN {X 0,Y 270.169,Z 228.452,A -85,B 0,C 180,E1 -17959.548,E2 -17959.548} C_VEL
LIN {X 0,Y 269.492,Z 228.533,A -85,B 0,C 180,E1 -17960.793,E2 -17960.793} C_VEL
LIN {X 0,Y 266.704,Z 228.889,A -85,B 0,C 180,E1 -17962.824,E2 -17962.824} C_VEL
LIN {X 0,Y 263.509,Z 229.292,A -85,B 0,C 180,E1 -17965.322,E2 -17965.322} C_VEL
LIN {X 0,Y 263.154,Z 229.323,A -85,B 0,C 180,E1 -17966.186,E2 -17966.186} C_VEL
LIN {X 0,Y 263.146,Z 229.302,A -85,B 0,C 180,E1 -17969.506,E2 -17969.506} C_VEL
LIN {X 0,Y 263.189,Z 229.32,A -85,B 0,C 180,E1 -17973.002,E2 -17973.002} C_VEL
LIN {X 0,Y 263.179,Z 229.324,A -85,B 0,C 180,E1 -17976.386,E2 -17976.386} C_VEL
LIN {X 0,Y 263.259,Z 229.317,A -85,B 0,C 180,E1 -17979.693,E2 -17979.693} C_VEL
LIN {X 0,Y 263.34,Z 229.303,A -85,B 0,C 180,E1 -17984.521,E2 -17984.521} C_VEL
LIN {X 0,Y 263.368,Z 229.296,A -85,B 0,C 180,E1 -17989.234,E2 -17989.234} C_VEL
LIN {X 0,Y 263.564,Z 229.28,A -85,B 0,C 180,E1 -17992.338,E2 -17992.338} C_VEL
LIN {X 0,Y 263.746,Z 229.248,A -85,B 0,C 180,E1 -17998.473,E2 -17998.473} C_VEL
LIN {X 0,Y 263.746,Z 229.257,A -85,B 0,C 180,E1 -18001.527,E2 -18001.527} C_VEL
LIN {X 0,Y 263.552,Z 229.275,A -85,B 0,C 180,E1 -18007.662,E2 -18007.662} C_VEL
LIN {X 0,Y 263.349,Z 229.31,A -85,B 0,C 180,E1 -18010.766,E2 -18010.766} C_VEL
LIN {X 0,Y 263.339,Z 229.31,A -85,B 0,C 180,E1 -18015.479,E2 -18015.479} C_VEL
LIN {X 0,Y 263.258,Z 229.317,A -85,B 0,C 180,E1 -18020.307,E2 -18020.307} C_VEL
LIN {X 0,Y 263.204,Z 229.316,A -85,B 0,C 180,E1 -18025.292,E2 -18025.292} C_VEL
LIN {X 0,Y 263.175,Z 229.329,A -85,B 0,C 180,E1 -18028.73,E2 -18028.73} C_VEL
LIN {X 0,Y 263.129,Z 229.326,A -85,B 0,C 180,E1 -18032.289,E2 -18032.289} C_VEL
LIN {X 0,Y 263.16,Z 229.322,A -85,B 0,C 180,E1 -18035.982,E2 -18035.982} C_VEL
LIN {X 0,Y 263.144,Z 229.401,A -85,B 0,C 180,E1 -18040.365,E2 -18040.365} C_VEL
LIN {X 0,Y 265.404,Z 236.51,A -85,B 0,C 180,E1 -18043.445,E2 -18043.445} C_VEL
LIN {X 0,Y 268.622,Z 241.567,A -85,B 0,C 180,E1 -18044.35,E2 -18044.35} C_VEL
LIN {X 0,Y 275.753,Z 253.315,A -85,B 0,C 180,E1 -18046.252,E2 -18046.252} C_VEL
LIN {X 0,Y 282.843,Z 266.322,A -85,B 0,C 180,E1 -18048.038,E2 -18048.038} C_VEL
LIN {X 0,Y 289.558,Z 279.832,A -85,B 0,C 180,E1 -18049.646,E2 -18049.646} C_VEL
LIN {X 0,Y 296.393,Z 295.692,A -85,B 0,C 180,E1 -18051.236,E2 -18051.236} C_VEL
LIN {X 0,Y 296.832,Z 298.302,A -85,B 0,C 180,E1 -18051.382,E2 -18051.382} C_VEL
LIN {X 0,Y 292.4,Z 399.015,A -85,B 0,C 180,E1 -18053.764,E2 -18053.764} C_VEL
LIN {X 0,Y 291.178,Z 414.326,A -85,B 0,C 180,E1 -18054.283,E2 -18054.283} C_VEL
LIN {X 0,Y 289.215,Z 429.884,A -85,B 0,C 180,E1 -18055.071,E2 -18055.071} C_VEL
LIN {X 0,Y 287.117,Z 442.773,A -85,B 0,C 180,E1 -18055.95,E2 -18055.95} C_VEL
LIN {X 0,Y 284.643,Z 455.846,A -85,B 0,C 180,E1 -18057.1,E2 -18057.1} C_VEL
LIN {X 0,Y 281.632,Z 469.432,A -85,B 0,C 180,E1 -18058.606,E2 -18058.606} C_VEL
LIN {X 0,Y 278.137,Z 482.991,A -85,B 0,C 180,E1 -18060.481,E2 -18060.481} C_VEL
LIN {X 0,Y 274.812,Z 495.202,A -85,B 0,C 180,E1 -18062.592,E2 -18062.592} C_VEL
LIN {X 0,Y 271.554,Z 506.252,A -85,B 0,C 180,E1 -18064.934,E2 -18064.934} C_VEL
LIN {X 0,Y 268.95,Z 515.484,A -85,B 0,C 180,E1 -18067.33,E2 -18067.33} C_VEL
LIN {X 0,Y 266.394,Z 523.814,A -85,B 0,C 180,E1 -18069.943,E2 -18069.943} C_VEL
LIN {X 0,Y 264.229,Z 531.649,A -85,B 0,C 180,E1 -18072.988,E2 -18072.988} C_VEL
LIN {X 0,Y 262.695,Z 537.888,A -85,B 0,C 180,E1 -18076.068,E2 -18076.068} C_VEL
LIN {X 0,Y 261.66,Z 542.718,A -85,B 0,C 180,E1 -18079.163,E2 -18079.163} C_VEL
LIN {X 0,Y 261.15,Z 546.262,A -85,B 0,C 180,E1 -18082.267,E2 -18082.267} C_VEL
LIN {X 0,Y 261.017,Z 548.597,A -85,B 0,C 180,E1 -18085.367,E2 -18085.367} C_VEL
LIN {X 0,Y 261.108,Z 549.774,A -85,B 0,C 180,E1 -18088.458,E2 -18088.458} C_VEL
LIN {X 0,Y 261.108,Z 549.77,A -85,B 0,C 180,E1 -18091.542,E2 -18091.542} C_VEL
LIN {X 0,Y 261.084,Z 548.31,A -85,B 0,C 180,E1 -18095.137,E2 -18095.137} C_VEL
LIN {X 0,Y 261.15,Z 546.229,A -85,B 0,C 180,E1 -18097.733,E2 -18097.733} C_VEL
LIN {X 0,Y 261.66,Z 542.676,A -85,B 0,C 180,E1 -18100.837,E2 -18100.837} C_VEL
LIN {X 0,Y 262.684,Z 537.834,A -85,B 0,C 180,E1 -18103.933,E2 -18103.933} C_VEL
LIN {X 0,Y 264.155,Z 531.569,A -85,B 0,C 180,E1 -18107.017,E2 -18107.017} C_VEL
LIN {X 0,Y 266.386,Z 523.715,A -85,B 0,C 180,E1 -18110.058,E2 -18110.058} C_VEL
LIN {X 0,Y 268.944,Z 515.371,A -85,B 0,C 180,E1 -18112.671,E2 -18112.671} C_VEL
LIN {X 0,Y 271.85,Z 505.133,A -85,B 0,C 180,E1 -18115.295,E2 -18115.295} C_VEL
LIN {X 0,Y 274.793,Z 495.049,A -85,B 0,C 180,E1 -18117.41,E2 -18117.41} C_VEL
LIN {X 0,Y 278.134,Z 482.811,A -85,B 0,C 180,E1 -18119.52,E2 -18119.52} C_VEL
LIN {X 0,Y 281.633,Z 469.189,A -85,B 0,C 180,E1 -18121.393,E2 -18121.393} C_VEL
LIN {X 0,Y 284.706,Z 455.172,A -85,B 0,C 180,E1 -18122.935,E2 -18122.935} C_VEL
LIN {X 0,Y 287.291,Z 441.379,A -85,B 0,C 180,E1 -18124.132,E2 -18124.132} C_VEL
LIN {X 0,Y 289.348,Z 428.13,A -85,B 0,C 180,E1 -18125.017,E2 -18125.017} C_VEL
LIN {X 0,Y 291.165,Z 413.681,A -85,B 0,C 180,E1 -18125.719,E2 -18125.719} C_VEL
LIN {X 0,Y 292.292,Z 399.436,A -85,B 0,C 180,E1 -18126.198,E2 -18126.198} C_VEL
LIN {X 0,Y 296.742,Z 299.622,A -85,B 0,C 180,E1 -18128.552,E2 -18128.552} C_VEL
LIN {X 0,Y 296.272,Z 295.447,A -85,B 0,C 180,E1 -18128.75,E2 -18128.75} C_VEL
LIN {X 0,Y 288.692,Z 278.055,A -85,B 0,C 180,E1 -18130.512,E2 -18130.512} C_VEL
LIN {X 0,Y 281.052,Z 262.943,A -85,B 0,C 180,E1 -18132.353,E2 -18132.353} C_VEL
LIN {X 0,Y 274.108,Z 250.605,A -85,B 0,C 180,E1 -18134.118,E2 -18134.118} C_VEL
LIN {X 0,Y 267.85,Z 240.548,A -85,B 0,C 180,E1 -18135.797,E2 -18135.797} C_VEL
LIN {X 0,Y 265.346,Z 236.304,A -85,B 0,C 180,E1 -18136.543,E2 -18136.543} C_VEL
LIN {X 0,Y 263.159,Z 229.321,A -85,B 0,C 180,E1 -18139.637,E2 -18139.637} C_VEL
LIN {X 0,Y 263.2,Z 229.32,A -85,B 0,C 180,E1 -18143.23,E2 -18143.23} C_VEL
LIN {X 0,Y 263.18,Z 229.322,A -85,B 0,C 180,E1 -18145.89,E2 -18145.89} C_VEL
LIN {X 0,Y 263.148,Z 229.323,A -85,B 0,C 180,E1 -18149.507,E2 -18149.507} C_VEL
LIN {X 0,Y 263.189,Z 229.318,A -85,B 0,C 180,E1 -18153.002,E2 -18153.002} C_VEL
LIN {X 0,Y 263.149,Z 229.315,A -85,B 0,C 180,E1 -18156.384,E2 -18156.384} C_VEL
LIN {X 0,Y 263.257,Z 229.292,A -85,B 0,C 180,E1 -18159.693,E2 -18159.693} C_VEL
LIN {X 0,Y 263.339,Z 229.303,A -85,B 0,C 180,E1 -18164.521,E2 -18164.521} C_VEL
LIN {X 0,Y 263.349,Z 229.306,A -85,B 0,C 180,E1 -18169.234,E2 -18169.234} C_VEL
LIN {X 0,Y 263.552,Z 229.274,A -85,B 0,C 180,E1 -18172.338,E2 -18172.338} C_VEL
LIN {X 0,Y 263.746,Z 229.256,A -85,B 0,C 180,E1 -18178.473,E2 -18178.473} C_VEL
LIN {X 0,Y 263.746,Z 229.254,A -85,B 0,C 180,E1 -18181.527,E2 -18181.527} C_VEL
LIN {X 0,Y 263.553,Z 229.275,A -85,B 0,C 180,E1 -18187.662,E2 -18187.662} C_VEL
LIN {X 0,Y 263.35,Z 229.307,A -85,B 0,C 180,E1 -18190.767,E2 -18190.767} C_VEL
LIN {X 0,Y 263.339,Z 229.305,A -85,B 0,C 180,E1 -18195.479,E2 -18195.479} C_VEL
LIN {X 0,Y 263.258,Z 229.31,A -85,B 0,C 180,E1 -18200.307,E2 -18200.307} C_VEL
LIN {X 0,Y 263.188,Z 229.294,A -85,B 0,C 180,E1 -18205.294,E2 -18205.294} C_VEL
LIN {X 0,Y 263.176,Z 229.325,A -85,B 0,C 180,E1 -18208.73,E2 -18208.73} C_VEL
LIN {X 0,Y 263.129,Z 229.333,A -85,B 0,C 180,E1 -18212.289,E2 -18212.289} C_VEL
LIN {X 0,Y 263.179,Z 229.319,A -85,B 0,C 180,E1 -18216.764,E2 -18216.764} C_VEL
LIN {X 0,Y 263.122,Z 229.327,A -85,B 0,C 180,E1 -18221.594,E2 -18221.594} C_VEL
LIN {X 0,Y 263.139,Z 229.46,A -85,B 0,C 180,E1 -18223.156,E2 -18223.156} C_VEL
LIN {X 0,Y 264.166,Z 232.264,A -85,B 0,C 180,E1 -18223.504,E2 -18223.504} C_VEL
LIN {X 0,Y 266.482,Z 234.818,A -85,B 0,C 180,E1 -18224.128,E2 -18224.128} C_VEL
LIN {X 0,Y 268.527,Z 238.035,A -85,B 0,C 180,E1 -18224.699,E2 -18224.699} C_VEL
LIN {X 0,Y 270.015,Z 240.052,A -85,B 0,C 180,E1 -18225.095,E2 -18225.095} C_VEL
LIN {X 0,Y 278.184,Z 252.007,A -85,B 0,C 180,E1 -18227.176,E2 -18227.176} C_VEL
LIN {X 0,Y 284.227,Z 261.86,A -85,B 0,C 180,E1 -18228.63,E2 -18228.63} C_VEL
LIN {X 0,Y 292.584,Z 278.321,A -85,B 0,C 180,E1 -18230.583,E2 -18230.583} C_VEL
LIN {X 0,Y 297.059,Z 288.385,A -85,B 0,C 180,E1 -18231.6,E2 -18231.6} C_VEL
LIN {X 0,Y 293.984,Z 360.141,A -85,B 0,C 180,E1 -18233.299,E2 -18233.299} C_VEL
LIN {X 0,Y 292.413,Z 391.858,A -85,B 0,C 180,E1 -18234.085,E2 -18234.085} C_VEL
LIN {X 0,Y 291.051,Z 406.659,A -85,B 0,C 180,E1 -18234.69,E2 -18234.69} C_VEL
LIN {X 0,Y 289.153,Z 421.784,A -85,B 0,C 180,E1 -18235.592,E2 -18235.592} C_VEL
LIN {X 0,Y 287.01,Z 435.182,A -85,B 0,C 180,E1 -18236.648,E2 -18236.648} C_VEL
LIN {X 0,Y 284.21,Z 449.544,A -85,B 0,C 180,E1 -18238.092,E2 -18238.092} C_VEL
LIN {X 0,Y 281.064,Z 462.995,A -85,B 0,C 180,E1 -18239.787,E2 -18239.787} C_VEL
LIN {X 0,Y 277.856,Z 475.2,A -85,B 0,C 180,E1 -18241.69,E2 -18241.69} C_VEL
LIN {X 0,Y 274.745,Z 486.583,A -85,B 0,C 180,E1 -18243.882,E2 -18243.882} C_VEL
LIN {X 0,Y 271.572,Z 497.104,A -85,B 0,C 180,E1 -18246.352,E2 -18246.352} C_VEL
LIN {X 0,Y 268.848,Z 506.057,A -85,B 0,C 180,E1 -18248.935,E2 -18248.935} C_VEL
LIN {X 0,Y 266.213,Z 514.332,A -85,B 0,C 180,E1 -18251.879,E2 -18251.879} C_VEL
LIN {X 0,Y 264.52,Z 520.402,A -85,B 0,C 180,E1 -18254.592,E2 -18254.592} C_VEL
LIN {X 0,Y 262.972,Z 525.842,A -85,B 0,C 180,E1 -18257.655,E2 -18257.655} C_VEL
LIN {X 0,Y 262.027,Z 529.942,A -85,B 0,C 180,E1 -18260.739,E2 -18260.739} C_VEL
LIN {X 0,Y 261.44,Z 532.821,A -85,B 0,C 180,E1 -18263.827,E2 -18263.827} C_VEL
LIN {X 0,Y 261.22,Z 534.548,A -85,B 0,C 180,E1 -18266.916,E2 -18266.916} C_VEL
LIN {X 0,Y 261.133,Z 535.151,A -85,B 0,C 180,E1 -18270,E2 -18270} C_VEL
LIN {X 0,Y 261.217,Z 534.588,A -85,B 0,C 180,E1 -18273.084,E2 -18273.084} C_VEL
LIN {X 0,Y 261.438,Z 532.914,A -85,B 0,C 180,E1 -18276.173,E2 -18276.173} C_VEL
LIN {X 0,Y 262.003,Z 530.084,A -85,B 0,C 180,E1 -18279.261,E2 -18279.261} C_VEL
LIN {X 0,Y 262.955,Z 526.031,A -85,B 0,C 180,E1 -18282.346,E2 -18282.346} C_VEL
LIN {X 0,Y 264.495,Z 520.65,A -85,B 0,C 180,E1 -18285.409,E2 -18285.409} C_VEL
LIN {X 0,Y 266.472,Z 513.793,A -85,B 0,C 180,E1 -18288.45,E2 -18288.45} C_VEL
LIN {X 0,Y 268.738,Z 506.416,A -85,B 0,C 180,E1 -18291.074,E2 -18291.074} C_VEL
LIN {X 0,Y 271.463,Z 497.52,A -85,B 0,C 180,E1 -18293.658,E2 -18293.658} C_VEL
LIN {X 0,Y 274.235,Z 488.443,A -85,B 0,C 180,E1 -18295.827,E2 -18295.827} C_VEL
LIN {X 0,Y 276.686,Z 479.678,A -85,B 0,C 180,E1 -18297.616,E2 -18297.616} C_VEL
LIN {X 0,Y 279.802,Z 468.374,A -85,B 0,C 180,E1 -18299.533,E2 -18299.533} C_VEL
LIN {X 0,Y 282.789,Z 456.087,A -85,B 0,C 180,E1 -18301.251,E2 -18301.251} C_VEL
LIN {X 0,Y 285.678,Z 442.646,A -85,B 0,C 180,E1 -18302.766,E2 -18302.766} C_VEL
LIN {X 0,Y 288.093,Z 429.129,A -85,B 0,C 180,E1 -18303.98,E2 -18303.98} C_VEL
LIN {X 0,Y 290.227,Z 414.401,A -85,B 0,C 180,E1 -18305.001,E2 -18305.001} C_VEL
LIN {X 0,Y 291.833,Z 399.88,A -85,B 0,C 180,E1 -18305.731,E2 -18305.731} C_VEL
LIN {X 0,Y 292.937,Z 385.423,A -85,B 0,C 180,E1 -18306.212,E2 -18306.212} C_VEL
LIN {X 0,Y 296.305,Z 308.442,A -85,B 0,C 180,E1 -18308.038,E2 -18308.038} C_VEL
LIN {X 0,Y 297.193,Z 288.538,A -85,B 0,C 180,E1 -18308.505,E2 -18308.505} C_VEL
LIN {X 0,Y 289.659,Z 272.249,A -85,B 0,C 180,E1 -18310.226,E2 -18310.226} C_VEL
LIN {X 0,Y 282.176,Z 258.16,A -85,B 0,C 180,E1 -18312.004,E2 -18312.004} C_VEL
LIN {X 0,Y 274.225,Z 246.151,A -85,B 0,C 180,E1 -18313.955,E2 -18313.955} C_VEL
LIN {X 0,Y 268.987,Z 238.519,A -85,B 0,C 180,E1 -18315.332,E2 -18315.332} C_VEL
LIN {X 0,Y 266.693,Z 235.305,A -85,B 0,C 180,E1 -18315.958,E2 -18315.958} C_VEL
LIN {X 0,Y 265.865,Z 234.08,A -85,B 0,C 180,E1 -18316.191,E2 -18316.191} C_VEL
LIN {X 0,Y 263.954,Z 231.819,A -85,B 0,C 180,E1 -18316.716,E2 -18316.716} C_VEL
LIN {X 0,Y 263.122,Z 229.316,A -85,B 0,C 180,E1 -18317.037,E2 -18317.037} C_VEL
LIN {X 0,Y 263.134,Z 229.323,A -85,B 0,C 180,E1 -18320.763,E2 -18320.763} C_VEL
LIN {X 0,Y 263.185,Z 229.31,A -85,B 0,C 180,E1 -18324.021,E2 -18324.021} C_VEL
LIN {X 0,Y 263.154,Z 229.323,A -85,B 0,C 180,E1 -18326.186,E2 -18326.186} C_VEL
LIN {X 0,Y 262.43,Z 229.396,A -85,B 0,C 180,E1 -18327.463,E2 -18327.463} C_VEL
LIN {X 0,Y 259.583,Z 229.756,A -85,B 0,C 180,E1 -18329.547,E2 -18329.547} C_VEL
LIN {X 0,Y 257.204,Z 230.068,A -85,B 0,C 180,E1 -18331.242,E2 -18331.242} C_VEL
LIN {X 0,Y 256.188,Z 230.196,A -85,B 0,C 180,E1 -18332.555,E2 -18332.555} C_VEL
LIN {X 0,Y 256.106,Z 230.201,A -85,B 0,C 180,E1 -18333,E2 -18333} C_VEL
LIN {X 0,Y 256.163,Z 230.202,A -85,B 0,C 180,E1 -18335.698,E2 -18335.698} C_VEL
LIN {X 0,Y 256.162,Z 230.201,A -85,B 0,C 180,E1 -18339.104,E2 -18339.104} C_VEL
LIN {X 0,Y 256.29,Z 230.186,A -85,B 0,C 180,E1 -18344.084,E2 -18344.084} C_VEL
LIN {X 0,Y 256.304,Z 230.178,A -85,B 0,C 180,E1 -18348.934,E2 -18348.934} C_VEL
LIN {X 0,Y 256.532,Z 230.155,A -85,B 0,C 180,E1 -18352.127,E2 -18352.127} C_VEL
LIN {X 0,Y 256.709,Z 230.125,A -85,B 0,C 180,E1 -18358.431,E2 -18358.431} C_VEL
LIN {X 0,Y 256.709,Z 230.133,A -85,B 0,C 180,E1 -18361.569,E2 -18361.569} C_VEL
LIN {X 0,Y 256.475,Z 230.164,A -85,B 0,C 180,E1 -18366.293,E2 -18366.293} C_VEL
LIN {X 0,Y 256.421,Z 230.162,A -85,B 0,C 180,E1 -18369.465,E2 -18369.465} C_VEL
LIN {X 0,Y 256.245,Z 230.188,A -85,B 0,C 180,E1 -18374.291,E2 -18374.291} C_VEL
LIN {X 0,Y 256.199,Z 230.187,A -85,B 0,C 180,E1 -18377.563,E2 -18377.563} C_VEL
LIN {X 0,Y 256.152,Z 230.195,A -85,B 0,C 180,E1 -18381.12,E2 -18381.12} C_VEL
LIN {X 0,Y 256.184,Z 230.191,A -85,B 0,C 180,E1 -18385.139,E2 -18385.139} C_VEL
LIN {X 0,Y 256.109,Z 230.21,A -85,B 0,C 180,E1 -18389.6,E2 -18389.6} C_VEL
LIN {X 0,Y 256.072,Z 230.204,A -85,B 0,C 180,E1 -18393.292,E2 -18393.292} C_VEL
LIN {X 0,Y 256.113,Z 230.204,A -85,B 0,C 180,E1 -18397.272,E2 -18397.272} C_VEL
LIN {X 0,Y 256.086,Z 230.3,A -85,B 0,C 180,E1 -18398.95,E2 -18398.95} C_VEL
LIN {X 0,Y 258.123,Z 236.397,A -85,B 0,C 180,E1 -18401.717,E2 -18401.717} C_VEL
LIN {X 0,Y 261.13,Z 241.079,A -85,B 0,C 180,E1 -18402.633,E2 -18402.633} C_VEL
LIN {X 0,Y 268.755,Z 253.324,A -85,B 0,C 180,E1 -18404.815,E2 -18404.815} C_VEL
LIN {X 0,Y 275.685,Z 265.439,A -85,B 0,C 180,E1 -18406.664,E2 -18406.664} C_VEL
LIN {X 0,Y 283.659,Z 281.353,A -85,B 0,C 180,E1 -18408.682,E2 -18408.682} C_VEL
LIN {X 0,Y 291.141,Z 298.658,A -85,B 0,C 180,E1 -18410.499,E2 -18410.499} C_VEL
LIN {X 0,Y 291.124,Z 303.997,A -85,B 0,C 180,E1 -18410.663,E2 -18410.663} C_VEL
LIN {X 0,Y 286.406,Z 403.335,A -85,B 0,C 180,E1 -18413.045,E2 -18413.045} C_VEL
LIN {X 0,Y 284.94,Z 418.711,A -85,B 0,C 180,E1 -18413.65,E2 -18413.65} C_VEL
LIN {X 0,Y 282.783,Z 433.596,A -85,B 0,C 180,E1 -18414.484,E2 -18414.484} C_VEL
LIN {X 0,Y 280.508,Z 446.56,A -85,B 0,C 180,E1 -18415.47,E2 -18415.47} C_VEL
LIN {X 0,Y 277.714,Z 460.313,A -85,B 0,C 180,E1 -18416.806,E2 -18416.806} C_VEL
LIN {X 0,Y 274.572,Z 473.147,A -85,B 0,C 180,E1 -18418.351,E2 -18418.351} C_VEL
LIN {X 0,Y 271.354,Z 484.94,A -85,B 0,C 180,E1 -18420.095,E2 -18420.095} C_VEL
LIN {X 0,Y 267.909,Z 496.792,A -85,B 0,C 180,E1 -18422.25,E2 -18422.25} C_VEL
LIN {X 0,Y 264.887,Z 506.676,A -85,B 0,C 180,E1 -18424.434,E2 -18424.434} C_VEL
LIN {X 0,Y 261.94,Z 516.542,A -85,B 0,C 180,E1 -18427.106,E2 -18427.106} C_VEL
LIN {X 0,Y 259.337,Z 524.696,A -85,B 0,C 180,E1 -18429.787,E2 -18429.787} C_VEL
LIN {X 0,Y 257,Z 532.82,A -85,B 0,C 180,E1 -18433.16,E2 -18433.16} C_VEL
LIN {X 0,Y 255.421,Z 539.013,A -85,B 0,C 180,E1 -18436.475,E2 -18436.475} C_VEL
LIN {X 0,Y 254.613,Z 542.516,A -85,B 0,C 180,E1 -18438.86,E2 -18438.86} C_VEL
LIN {X 0,Y 254.087,Z 546.061,A -85,B 0,C 180,E1 -18442.051,E2 -18442.051} C_VEL
LIN {X 0,Y 253.932,Z 548.397,A -85,B 0,C 180,E1 -18445.237,E2 -18445.237} C_VEL
LIN {X 0,Y 254.013,Z 549.573,A -85,B 0,C 180,E1 -18448.415,E2 -18448.415} C_VEL
LIN {X 0,Y 254.053,Z 549.728,A -85,B 0,C 180,E1 -18450,E2 -18450} C_VEL
LIN {X 0,Y 253.936,Z 549.115,A -85,B 0,C 180,E1 -18453.173,E2 -18453.173} C_VEL
LIN {X 0,Y 253.957,Z 547.348,A -85,B 0,C 180,E1 -18456.355,E2 -18456.355} C_VEL
LIN {X 0,Y 254.313,Z 544.405,A -85,B 0,C 180,E1 -18459.544,E2 -18459.544} C_VEL
LIN {X 0,Y 255.109,Z 540.22,A -85,B 0,C 180,E1 -18462.732,E2 -18462.732} C_VEL
LIN {X 0,Y 256.406,Z 534.683,A -85,B 0,C 180,E1 -18465.908,E2 -18465.908} C_VEL
LIN {X 0,Y 258.408,Z 527.65,A -85,B 0,C 180,E1 -18469.048,E2 -18469.048} C_VEL
LIN {X 0,Y 261.081,Z 518.909,A -85,B 0,C 180,E1 -18472.139,E2 -18472.139} C_VEL
LIN {X 0,Y 263.581,Z 511.08,A -85,B 0,C 180,E1 -18474.411,E2 -18474.411} C_VEL
LIN {X 0,Y 266.372,Z 501.841,A -85,B 0,C 180,E1 -18476.649,E2 -18476.649} C_VEL
LIN {X 0,Y 269.561,Z 490.962,A -85,B 0,C 180,E1 -18478.837,E2 -18478.837} C_VEL
LIN {X 0,Y 272.9,Z 479.095,A -85,B 0,C 180,E1 -18480.786,E2 -18480.786} C_VEL
LIN {X 0,Y 276.192,Z 466.445,A -85,B 0,C 180,E1 -18482.467,E2 -18482.467} C_VEL
LIN {X 0,Y 279.059,Z 453.553,A -85,B 0,C 180,E1 -18483.862,E2 -18483.862} C_VEL
LIN {X 0,Y 281.608,Z 440.041,A -85,B 0,C 180,E1 -18485.029,E2 -18485.029} C_VEL
LIN {X 0,Y 283.889,Z 425.852,A -85,B 0,C 180,E1 -18485.957,E2 -18485.957} C_VEL
LIN {X 0,Y 285.735,Z 410.56,A -85,B 0,C 180,E1 -18486.671,E2 -18486.671} C_VEL
LIN {X 0,Y 286.843,Z 394.44,A -85,B 0,C 180,E1 -18487.164,E2 -18487.164} C_VEL
LIN {X 0,Y 291.157,Z 299.544,A -85,B 0,C 180,E1 -18489.428,E2 -18489.428} C_VEL
LIN {X 0,Y 290.27,Z 296.709,A -85,B 0,C 180,E1 -18489.66,E2 -18489.66} C_VEL
LIN {X 0,Y 282.98,Z 279.999,A -85,B 0,C 180,E1 -18491.435,E2 -18491.435} C_VEL
LIN {X 0,Y 275.29,Z 264.82,A -85,B 0,C 180,E1 -18493.382,E2 -18493.382} C_VEL
LIN {X 0,Y 267.708,Z 251.534,A -85,B 0,C 180,E1 -18495.417,E2 -18495.417} C_VEL
LIN {X 0,Y 260.699,Z 240.558,A -85,B 0,C 180,E1 -18497.424,E2 -18497.424} C_VEL
LIN {X 0,Y 258.017,Z 236.048,A -85,B 0,C 180,E1 -18498.273,E2 -18498.273} C_VEL
LIN {X 0,Y 256.101,Z 230.2,A -85,B 0,C 180,E1 -18501.114,E2 -18501.114} C_VEL
LIN {X 0,Y 256.117,Z 230.196,A -85,B 0,C 180,E1 -18504.813,E2 -18504.813} C_VEL
LIN {X 0,Y 256.089,Z 230.207,A -85,B 0,C 180,E1 -18508.572,E2 -18508.572} C_VEL
LIN {X 0,Y 256.14,Z 230.2,A -85,B 0,C 180,E1 -18512.196,E2 -18512.196} C_VEL
LIN {X 0,Y 256.137,Z 230.2,A -85,B 0,C 180,E1 -18515.696,E2 -18515.696} C_VEL
LIN {X 0,Y 256.156,Z 230.17,A -85,B 0,C 180,E1 -18519.104,E2 -18519.104} C_VEL
LIN {X 0,Y 256.289,Z 230.178,A -85,B 0,C 180,E1 -18524.085,E2 -18524.085} C_VEL
LIN {X 0,Y 256.288,Z 230.177,A -85,B 0,C 180,E1 -18527.328,E2 -18527.328} C_VEL
LIN {X 0,Y 256.509,Z 230.15,A -85,B 0,C 180,E1 -18532.126,E2 -18532.126} C_VEL
LIN {X 0,Y 256.493,Z 230.155,A -85,B 0,C 180,E1 -18536.859,E2 -18536.859} C_VEL
LIN {X 0,Y 256.76,Z 230.116,A -85,B 0,C 180,E1 -18540,E2 -18540} C_VEL
LIN {X 0,Y 256.493,Z 230.155,A -85,B 0,C 180,E1 -18543.142,E2 -18543.142} C_VEL
LIN {X 0,Y 256.51,Z 230.15,A -85,B 0,C 180,E1 -18547.874,E2 -18547.874} C_VEL
LIN {X 0,Y 256.288,Z 230.176,A -85,B 0,C 180,E1 -18552.673,E2 -18552.673} C_VEL
LIN {X 0,Y 256.256,Z 230.182,A -85,B 0,C 180,E1 -18556.285,E2 -18556.285} C_VEL
LIN {X 0,Y 256.157,Z 230.194,A -85,B 0,C 180,E1 -18560.896,E2 -18560.896} C_VEL
LIN {X 0,Y 256.166,Z 230.169,A -85,B 0,C 180,E1 -18565.13,E2 -18565.13} C_VEL
LIN {X 0,Y 256.11,Z 230.208,A -85,B 0,C 180,E1 -18569.6,E2 -18569.6} C_VEL
LIN {X 0,Y 256.064,Z 230.208,A -85,B 0,C 180,E1 -18573.293,E2 -18573.293} C_VEL
LIN {X 0,Y 256.111,Z 230.2,A -85,B 0,C 180,E1 -18577.271,E2 -18577.271} C_VEL
LIN {X 0,Y 256.082,Z 230.275,A -85,B 0,C 180,E1 -18581.465,E2 -18581.465} C_VEL
LIN {X 0,Y 257.021,Z 232.95,A -85,B 0,C 180,E1 -18581.813,E2 -18581.813} C_VEL
LIN {X 0,Y 259.199,Z 235.246,A -85,B 0,C 180,E1 -18582.446,E2 -18582.446} C_VEL
LIN {X 0,Y 261.628,Z 239.022,A -85,B 0,C 180,E1 -18583.178,E2 -18583.178} C_VEL
LIN {X 0,Y 263.031,Z 240.772,A -85,B 0,C 180,E1 -18583.573,E2 -18583.573} C_VEL
LIN {X 0,Y 271.496,Z 253.013,A -85,B 0,C 180,E1 -18585.879,E2 -18585.879} C_VEL
LIN {X 0,Y 278.687,Z 264.369,A -85,B 0,C 180,E1 -18587.697,E2 -18587.697} C_VEL
LIN {X 0,Y 286.129,Z 278.9,A -85,B 0,C 180,E1 -18589.522,E2 -18589.522} C_VEL
LIN {X 0,Y 291.437,Z 290.498,A -85,B 0,C 180,E1 -18590.777,E2 -18590.777} C_VEL
LIN {X 0,Y 289.737,Z 330.255,A -85,B 0,C 180,E1 -18591.744,E2 -18591.744} C_VEL
LIN {X 0,Y 286.829,Z 390.926,A -85,B 0,C 180,E1 -18593.219,E2 -18593.219} C_VEL
LIN {X 0,Y 285.293,Z 406.87,A -85,B 0,C 180,E1 -18593.866,E2 -18593.866} C_VEL
LIN {X 0,Y 283.333,Z 421.992,A -85,B 0,C 180,E1 -18594.781,E2 -18594.781} C_VEL
LIN {X 0,Y 281.011,Z 435.947,A -85,B 0,C 180,E1 -18595.904,E2 -18595.904} C_VEL
LIN {X 0,Y 278.199,Z 449.75,A -85,B 0,C 180,E1 -18597.318,E2 -18597.318} C_VEL
LIN {X 0,Y 274.927,Z 463.2,A -85,B 0,C 180,E1 -18599.04,E2 -18599.04} C_VEL
LIN {X 0,Y 271.607,Z 475.405,A -85,B 0,C 180,E1 -18600.977,E2 -18600.977} C_VEL
LIN {X 0,Y 268.272,Z 487.03,A -85,B 0,C 180,E1 -18603.265,E2 -18603.265} C_VEL
LIN {X 0,Y 265.049,Z 497.308,A -85,B 0,C 180,E1 -18605.733,E2 -18605.733} C_VEL
LIN {X 0,Y 262.197,Z 506.262,A -85,B 0,C 180,E1 -18608.374,E2 -18608.374} C_VEL
LIN {X 0,Y 259.695,Z 513.681,A -85,B 0,C 180,E1 -18611.05,E2 -18611.05} C_VEL
LIN {X 0,Y 257.646,Z 520.605,A -85,B 0,C 180,E1 -18614.171,E2 -18614.171} C_VEL
LIN {X 0,Y 256.011,Z 526.045,A -85,B 0,C 180,E1 -18617.314,E2 -18617.314} C_VEL
LIN {X 0,Y 254.992,Z 530.145,A -85,B 0,C 180,E1 -18620.481,E2 -18620.481} C_VEL
LIN {X 0,Y 254.375,Z 533.023,A -85,B 0,C 180,E1 -18623.655,E2 -18623.655} C_VEL
LIN {X 0,Y 254.137,Z 534.749,A -85,B 0,C 180,E1 -18626.829,E2 -18626.829} C_VEL
LIN {X 0,Y 254.061,Z 535.352,A -85,B 0,C 180,E1 -18630,E2 -18630} C_VEL
LIN {X 0,Y 254.132,Z 534.789,A -85,B 0,C 180,E1 -18633.171,E2 -18633.171} C_VEL
LIN {X 0,Y 254.371,Z 533.114,A -85,B 0,C 180,E1 -18636.345,E2 -18636.345} C_VEL
LIN {X 0,Y 254.971,Z 530.285,A -85,B 0,C 180,E1 -18639.519,E2 -18639.519} C_VEL
LIN {X 0,Y 255.995,Z 526.231,A -85,B 0,C 180,E1 -18642.687,E2 -18642.687} C_VEL
LIN {X 0,Y 257.622,Z 520.851,A -85,B 0,C 180,E1 -18645.831,E2 -18645.831} C_VEL
LIN {X 0,Y 259.692,Z 513.994,A -85,B 0,C 180,E1 -18648.95,E2 -18648.95} C_VEL
LIN {X 0,Y 262.1,Z 506.616,A -85,B 0,C 180,E1 -18651.635,E2 -18651.635} C_VEL
LIN {X 0,Y 264.931,Z 497.72,A -85,B 0,C 180,E1 -18654.278,E2 -18654.278} C_VEL
LIN {X 0,Y 267.801,Z 488.643,A -85,B 0,C 180,E1 -18656.495,E2 -18656.495} C_VEL
LIN {X 0,Y 270.962,Z 477.933,A -85,B 0,C 180,E1 -18658.674,E2 -18658.674} C_VEL
LIN {X 0,Y 274.183,Z 466.236,A -85,B 0,C 180,E1 -18660.626,E2 -18660.626} C_VEL
LIN {X 0,Y 277.397,Z 453.455,A -85,B 0,C 180,E1 -18662.357,E2 -18662.357} C_VEL
LIN {X 0,Y 280.377,Z 439.664,A -85,B 0,C 180,E1 -18663.858,E2 -18663.858} C_VEL
LIN {X 0,Y 282.849,Z 425.59,A -85,B 0,C 180,E1 -18665.07,E2 -18665.07} C_VEL
LIN {X 0,Y 284.891,Z 410.958,A -85,B 0,C 180,E1 -18666.029,E2 -18666.029} C_VEL
LIN {X 0,Y 286.362,Z 397.069,A -85,B 0,C 180,E1 -18666.687,E2 -18666.687} C_VEL
LIN {X 0,Y 287.538,Z 380.715,A -85,B 0,C 180,E1 -18667.168,E2 -18667.168} C_VEL
LIN {X 0,Y 290.729,Z 309.197,A -85,B 0,C 180,E1 -18668.885,E2 -18668.885} C_VEL
LIN {X 0,Y 291.569,Z 290.726,A -85,B 0,C 180,E1 -18669.327,E2 -18669.327} C_VEL
LIN {X 0,Y 283.866,Z 274.138,A -85,B 0,C 180,E1 -18671.166,E2 -18671.166} C_VEL
LIN {X 0,Y 277.505,Z 262.323,A -85,B 0,C 180,E1 -18672.74,E2 -18672.74} C_VEL
LIN {X 0,Y 270.462,Z 251.509,A -85,B 0,C 180,E1 -18674.537,E2 -18674.537} C_VEL
LIN {X 0,Y 264.883,Z 243.455,A -85,B 0,C 180,E1 -18676.053,E2 -18676.053} C_VEL
LIN {X 0,Y 261.958,Z 239.363,A -85,B 0,C 180,E1 -18676.886,E2 -18676.886} C_VEL
LIN {X 0,Y 259.733,Z 236.116,A -85,B 0,C 180,E1 -18677.547,E2 -18677.547} C_VEL
LIN {X 0,Y 259.038,Z 235.124,A -85,B 0,C 180,E1 -18677.756,E2 -18677.756} C_VEL
LIN {X 0,Y 257.021,Z 232.945,A -85,B 0,C 180,E1 -18678.347,E2 -18678.347} C_VEL
LIN {X 0,Y 256.08,Z 230.197,A -85,B 0,C 180,E1 -18678.748,E2 -18678.748} C_VEL
LIN {X 0,Y 256.143,Z 230.177,A -85,B 0,C 180,E1 -18682.869,E2 -18682.869} C_VEL
LIN {X 0,Y 256.082,Z 230.194,A -85,B 0,C 180,E1 -18686.709,E2 -18686.709} C_VEL
LIN {X 0,Y 256.135,Z 230.203,A -85,B 0,C 180,E1 -18691.404,E2 -18691.404} C_VEL
LIN {X 0,Y 256.106,Z 230.201,A -85,B 0,C 180,E1 -18693,E2 -18693} C_VEL
LIN {X 0,Y 255.428,Z 230.287,A -85,B 0,C 180,E1 -18694.312,E2 -18694.312} C_VEL
LIN {X 0,Y 252.554,Z 230.646,A -85,B 0,C 180,E1 -18696.45,E2 -18696.45} C_VEL
LIN {X 0,Y 250.144,Z 230.944,A -85,B 0,C 180,E1 -18698.191,E2 -18698.191} C_VEL
LIN {X 0,Y 249.152,Z 231.075,A -85,B 0,C 180,E1 -18699.541,E2 -18699.541} C_VEL
LIN {X 0,Y 249.093,Z 231.077,A -85,B 0,C 180,E1 -18699.999,E2 -18699.999} C_VEL
LIN {X 0,Y 249.238,Z 231.064,A -85,B 0,C 180,E1 -18703.621,E2 -18703.621} C_VEL
LIN {X 0,Y 249.247,Z 231.06,A -85,B 0,C 180,E1 -18708.616,E2 -18708.616} C_VEL
LIN {X 0,Y 249.474,Z 231.033,A -85,B 0,C 180,E1 -18711.902,E2 -18711.902} C_VEL
LIN {X 0,Y 249.43,Z 231.04,A -85,B 0,C 180,E1 -18716.769,E2 -18716.769} C_VEL
LIN {X 0,Y 249.723,Z 230.991,A -85,B 0,C 180,E1 -18720,E2 -18720} C_VEL
LIN {X 0,Y 249.429,Z 231.03,A -85,B 0,C 180,E1 -18723.23,E2 -18723.23} C_VEL
LIN {X 0,Y 249.448,Z 231.04,A -85,B 0,C 180,E1 -18726.471,E2 -18726.471} C_VEL
LIN {X 0,Y 249.338,Z 231.047,A -85,B 0,C 180,E1 -18729.736,E2 -18729.736} C_VEL
LIN {X 0,Y 249.192,Z 231.071,A -85,B 0,C 180,E1 -18734.704,E2 -18734.704} C_VEL
LIN {X 0,Y 249.13,Z 231.07,A -85,B 0,C 180,E1 -18738.078,E2 -18738.078} C_VEL
LIN {X 0,Y 249.082,Z 231.075,A -85,B 0,C 180,E1 -18741.518,E2 -18741.518} C_VEL
LIN {X 0,Y 249.126,Z 231.069,A -85,B 0,C 180,E1 -18745.482,E2 -18745.482} C_VEL
LIN {X 0,Y 249.079,Z 231.085,A -85,B 0,C 180,E1 -18748.994,E2 -18748.994} C_VEL
LIN {X 0,Y 249.029,Z 231.081,A -85,B 0,C 180,E1 -18752.426,E2 -18752.426} C_VEL
LIN {X 0,Y 249.1,Z 231.076,A -85,B 0,C 180,E1 -18757.111,E2 -18757.111} C_VEL
LIN {X 0,Y 249.093,Z 231.104,A -85,B 0,C 180,E1 -18757.389,E2 -18757.389} C_VEL
LIN {X 0,Y 250.664,Z 236.001,A -85,B 0,C 180,E1 -18759.762,E2 -18759.762} C_VEL
LIN {X 0,Y 254.094,Z 241.118,A -85,B 0,C 180,E1 -18760.894,E2 -18760.894} C_VEL
LIN {X 0,Y 261.521,Z 252.907,A -85,B 0,C 180,E1 -18763.191,E2 -18763.191} C_VEL
LIN {X 0,Y 268.865,Z 265.352,A -85,B 0,C 180,E1 -18765.282,E2 -18765.282} C_VEL
LIN {X 0,Y 276.813,Z 280.857,A -85,B 0,C 180,E1 -18767.415,E2 -18767.415} C_VEL
LIN {X 0,Y 283.494,Z 295.782,A -85,B 0,C 180,E1 -18769.127,E2 -18769.127} C_VEL
LIN {X 0,Y 285.728,Z 301.173,A -85,B 0,C 180,E1 -18769.685,E2 -18769.685} C_VEL
LIN {X 0,Y 280.972,Z 400.155,A -85,B 0,C 180,E1 -18772.094,E2 -18772.094} C_VEL
LIN {X 0,Y 279.577,Z 415.778,A -85,B 0,C 180,E1 -18772.668,E2 -18772.668} C_VEL
LIN {X 0,Y 277.484,Z 430.8,A -85,B 0,C 180,E1 -18773.474,E2 -18773.474} C_VEL
LIN {X 0,Y 275.063,Z 444.372,A -85,B 0,C 180,E1 -18774.461,E2 -18774.461} C_VEL
LIN {X 0,Y 272.005,Z 459.088,A -85,B 0,C 180,E1 -18775.87,E2 -18775.87} C_VEL
LIN {X 0,Y 268.531,Z 472.949,A -85,B 0,C 180,E1 -18777.553,E2 -18777.553} C_VEL
LIN {X 0,Y 265.156,Z 484.74,A -85,B 0,C 180,E1 -18779.322,E2 -18779.322} C_VEL
LIN {X 0,Y 261.606,Z 496.592,A -85,B 0,C 180,E1 -18781.521,E2 -18781.521} C_VEL
LIN {X 0,Y 258.195,Z 507.188,A -85,B 0,C 180,E1 -18783.929,E2 -18783.929} C_VEL
LIN {X 0,Y 255.358,Z 516.341,A -85,B 0,C 180,E1 -18786.48,E2 -18786.48} C_VEL
LIN {X 0,Y 252.631,Z 524.495,A -85,B 0,C 180,E1 -18789.226,E2 -18789.226} C_VEL
LIN {X 0,Y 250.53,Z 531.245,A -85,B 0,C 180,E1 -18792.027,E2 -18792.027} C_VEL
LIN {X 0,Y 248.768,Z 537.484,A -85,B 0,C 180,E1 -18795.271,E2 -18795.271} C_VEL
LIN {X 0,Y 247.583,Z 542.314,A -85,B 0,C 180,E1 -18798.539,E2 -18798.539} C_VEL
LIN {X 0,Y 247.014,Z 545.859,A -85,B 0,C 180,E1 -18801.822,E2 -18801.822} C_VEL
LIN {X 0,Y 246.841,Z 548.25,A -85,B 0,C 180,E1 -18805.21,E2 -18805.21} C_VEL
LIN {X 0,Y 246.92,Z 549.372,A -85,B 0,C 180,E1 -18808.369,E2 -18808.369} C_VEL
LIN {X 0,Y 246.982,Z 549.528,A -85,B 0,C 180,E1 -18810,E2 -18810} C_VEL
LIN {X 0,Y 246.838,Z 548.914,A -85,B 0,C 180,E1 -18813.264,E2 -18813.264} C_VEL
LIN {X 0,Y 246.872,Z 547.146,A -85,B 0,C 180,E1 -18816.538,E2 -18816.538} C_VEL
LIN {X 0,Y 247.268,Z 544.202,A -85,B 0,C 180,E1 -18819.819,E2 -18819.819} C_VEL
LIN {X 0,Y 248.141,Z 540.017,A -85,B 0,C 180,E1 -18823.096,E2 -18823.096} C_VEL
LIN {X 0,Y 249.499,Z 534.478,A -85,B 0,C 180,E1 -18826.36,E2 -18826.36} C_VEL
LIN {X 0,Y 251.649,Z 527.446,A -85,B 0,C 180,E1 -18829.58,E2 -18829.58} C_VEL
LIN {X 0,Y 254.469,Z 518.704,A -85,B 0,C 180,E1 -18832.746,E2 -18832.746} C_VEL
LIN {X 0,Y 257.041,Z 510.874,A -85,B 0,C 180,E1 -18835.074,E2 -18835.074} C_VEL
LIN {X 0,Y 260.493,Z 499.995,A -85,B 0,C 180,E1 -18837.735,E2 -18837.735} C_VEL
LIN {X 0,Y 264.239,Z 487.769,A -85,B 0,C 180,E1 -18840.133,E2 -18840.133} C_VEL
LIN {X 0,Y 267.455,Z 476.535,A -85,B 0,C 180,E1 -18841.926,E2 -18841.926} C_VEL
LIN {X 0,Y 270.902,Z 463.416,A -85,B 0,C 180,E1 -18843.621,E2 -18843.621} C_VEL
LIN {X 0,Y 273.909,Z 449.806,A -85,B 0,C 180,E1 -18845.036,E2 -18845.036} C_VEL
LIN {X 0,Y 276.573,Z 435.313,A -85,B 0,C 180,E1 -18846.213,E2 -18846.213} C_VEL
LIN {X 0,Y 278.88,Z 420.3,A -85,B 0,C 180,E1 -18847.102,E2 -18847.102} C_VEL
LIN {X 0,Y 280.6,Z 404.634,A -85,B 0,C 180,E1 -18847.738,E2 -18847.738} C_VEL
LIN {X 0,Y 282.647,Z 363.964,A -85,B 0,C 180,E1 -18848.77,E2 -18848.77} C_VEL
LIN {X 0,Y 285.62,Z 301.126,A -85,B 0,C 180,E1 -18850.29,E2 -18850.29} C_VEL
LIN {X 0,Y 278.924,Z 285.396,A -85,B 0,C 180,E1 -18851.986,E2 -18851.986} C_VEL
LIN {X 0,Y 271.004,Z 269.412,A -85,B 0,C 180,E1 -18854.072,E2 -18854.072} C_VEL
LIN {X 0,Y 263.514,Z 256.167,A -85,B 0,C 180,E1 -18856.164,E2 -18856.164} C_VEL
LIN {X 0,Y 256.984,Z 245.762,A -85,B 0,C 180,E1 -18858.113,E2 -18858.113} C_VEL
LIN {X 0,Y 253.576,Z 240.472,A -85,B 0,C 180,E1 -18859.196,E2 -18859.196} C_VEL
LIN {X 0,Y 250.559,Z 235.734,A -85,B 0,C 180,E1 -18860.218,E2 -18860.218} C_VEL
LIN {X 0,Y 249.1,Z 231.072,A -85,B 0,C 180,E1 -18862.609,E2 -18862.609} C_VEL
LIN {X 0,Y 249.058,Z 231.08,A -85,B 0,C 180,E1 -18865.642,E2 -18865.642} C_VEL
